C03625=1096.715,71.531,441.280,176.195,16.215,152.221
C03626=1096.709,71.282,441.296,176.193,16.214,152.222
C03627=1096.703,71.032,441.313,176.190,16.213,152.222
C03628=1096.698,70.783,441.330,176.188,16.213,152.222
C03629=1096.692,70.534,441.346,176.185,16.211,152.223
C03630=1096.687,70.284,441.363,176.183,16.211,152.223
C03631=1096.681,70.035,441.380,176.180,16.210,152.223
C03632=1096.675,69.785,441.398,176.179,16.209,152.224
C03633=1096.669,69.536,441.414,176.176,16.209,152.224
C03634=1096.663,69.286,441.431,176.174,16.208,152.224
C03635=1096.657,69.037,441.448,176.172,16.207,152.225
C03636=1096.652,68.787,441.464,176.169,16.206,152.225
C03637=1096.646,68.538,441.481,176.167,16.205,152.225
C03638=1096.641,68.288,441.498,176.164,16.205,152.226
C03639=1096.635,68.039,441.514,176.162,16.204,152.226
C03640=1096.629,67.790,441.531,176.159,16.203,152.226
C03641=1096.623,67.541,441.548,176.157,16.202,152.227
C03642=1096.618,67.291,441.564,176.155,16.201,152.227
C03643=1096.612,67.042,441.581,176.152,16.201,152.227
C03644=1096.606,66.793,441.598,176.150,16.200,152.228
C03645=1096.601,66.543,441.615,176.148,16.199,152.228
C03646=1096.595,66.294,441.631,176.146,16.199,152.228
C03647=1096.590,66.044,441.648,176.143,16.197,152.228
C03648=1096.584,65.795,441.664,176.141,16.197,152.229
C03649=1096.578,65.546,441.680,176.138,16.196,152.229
C03650=1096.572,65.296,441.697,176.136,16.195,152.229
C03651=1096.566,65.047,441.714,176.133,16.194,152.230
C03652=1096.561,64.798,441.731,176.131,16.194,152.230
C03653=1096.555,64.548,441.747,176.129,16.192,152.230
C03654=1096.549,64.299,441.763,176.127,16.192,152.231
C03655=1096.543,64.024,441.782,176.124,16.191,152.231
C03656=1096.537,63.749,441.800,176.122,16.190,152.231
C03657=1096.531,63.475,441.818,176.119,16.189,152.232
C03658=1096.524,63.201,441.836,176.116,16.188,152.232
C03659=1096.519,62.952,441.853,176.114,16.187,152.232
C03660=1096.513,62.702,441.869,176.111,16.186,152.233
C03661=1096.507,62.453,441.885,176.109,16.186,152.233
C03662=1096.501,62.204,441.902,176.107,16.185,152.233
C03663=1096.495,61.954,441.918,176.105,16.184,152.234
C03664=1096.490,61.705,441.935,176.103,16.184,152.234
C03665=1096.484,61.455,441.951,176.100,16.182,152.234
C03666=1096.478,61.206,441.967,176.098,16.182,152.235
C03667=1096.472,60.957,441.983,176.095,16.181,152.235
C03668=1096.466,60.707,442.000,176.093,16.180,152.235
C03669=1096.461,60.458,442.017,176.091,16.179,152.235
C03670=1096.455,60.208,442.033,176.088,16.179,152.236
C03671=1096.449,59.959,442.049,176.086,16.178,152.236
C03672=1096.443,59.709,442.065,176.084,16.177,152.236
C03673=1096.437,59.460,442.082,176.082,16.176,152.237
C03674=1096.432,59.210,442.098,176.079,16.175,152.237
C03675=1096.426,58.961,442.115,176.077,16.174,152.237
C03676=1096.420,58.711,442.130,176.075,16.174,152.238
C03677=1096.414,58.462,442.146,176.072,16.172,152.238
C03678=1096.408,58.212,442.163,176.070,16.172,152.238
C03679=1096.403,57.964,442.179,176.068,16.171,152.239
C03680=1096.397,57.714,442.195,176.066,16.170,152.239
C03681=1096.391,57.465,442.212,176.063,16.169,152.239
C03682=1096.386,57.215,442.228,176.061,16.168,152.239
C03683=1096.380,56.966,442.244,176.059,16.168,152.240
C03684=1096.374,56.716,442.260,176.056,16.167,152.240
C03685=1096.368,56.467,442.276,176.054,16.166,152.240
C03686=1096.362,56.217,442.292,176.052,16.165,152.240
C03687=1096.356,55.968,442.309,176.050,16.164,152.241
C03688=1096.351,55.719,442.325,176.048,16.163,152.241
C03689=1096.346,55.469,442.341,176.045,16.162,152.241
C03690=1096.340,55.220,442.357,176.043,16.161,152.242
C03691=1096.334,54.970,442.373,176.040,16.161,152.242
C03692=1096.328,54.721,442.389,176.038,16.160,152.242
C03693=1096.322,54.472,442.406,176.036,16.159,152.242
C03694=1096.317,54.223,442.421,176.034,16.158,152.243
C03695=1096.311,53.973,442.437,176.032,16.157,152.243
C03696=1096.305,53.724,442.453,176.029,16.156,152.243
C03697=1096.299,53.474,442.469,176.027,16.155,152.244
C03698=1096.294,53.224,442.486,176.025,16.154,152.244
C03699=1096.288,52.975,442.502,176.023,16.153,152.244
C03700=1096.283,52.726,442.518,176.021,16.153,152.244
C03701=1096.277,52.476,442.533,176.018,16.151,152.245
C03702=1096.271,52.227,442.550,176.016,16.151,152.245
C03703=1096.265,51.978,442.566,176.014,16.149,152.245
C03704=1096.260,51.728,442.581,176.011,16.149,152.246
C03705=1096.254,51.479,442.597,176.010,16.148,152.246
C03706=1096.248,51.230,442.614,176.007,16.147,152.246
C03707=1096.243,50.980,442.629,176.005,16.146,152.246
C03708=1096.237,50.730,442.645,176.002,16.145,152.247
C03709=1096.232,50.481,442.661,176.000,16.144,152.247
C03710=1096.226,50.232,442.677,175.999,16.144,152.247
C03711=1096.220,49.982,442.693,175.996,16.142,152.247
C03712=1096.214,49.732,442.709,175.994,16.142,152.248
C03713=1096.209,49.484,442.724,175.991,16.140,152.248
C03714=1096.203,49.234,442.740,175.989,16.140,152.248
C03715=1096.197,48.984,442.756,175.988,16.139,152.248
C03716=1096.191,48.735,442.773,175.985,16.137,152.249
C03717=1096.186,48.486,442.788,175.983,16.137,152.249
C03718=1096.180,48.236,442.804,175.981,16.135,152.249
C03719=1096.174,47.961,442.822,175.979,16.135,152.249
C03720=1096.168,47.687,442.839,175.976,16.133,152.250
C03721=1096.162,47.412,442.857,175.973,16.132,152.250
C03722=1096.156,47.138,442.873,175.971,16.131,152.250
C03723=1096.150,46.888,442.889,175.969,16.130,152.250
C03724=1096.144,46.639,442.905,175.967,16.129,152.251
C03725=1096.139,46.389,442.921,175.965,16.129,152.251
C03726=1096.134,46.139,442.936,175.962,16.127,152.251
C03727=1096.128,45.890,442.952,175.960,16.127,152.251
C03728=1096.122,45.640,442.968,175.958,16.125,152.252
C03729=1096.117,45.391,442.984,175.956,16.125,152.252
C03730=1096.111,45.141,442.999,175.954,16.124,152.252
C03731=1096.105,44.892,443.015,175.951,16.122,152.252
C03732=1096.100,44.643,443.031,175.950,16.122,152.253
C03733=1096.094,44.393,443.047,175.948,16.121,152.253
C03734=1096.089,44.144,443.062,175.945,16.120,152.253
C03735=1096.083,43.894,443.078,175.943,16.119,152.253
C03736=1096.077,43.645,443.094,175.940,16.118,152.254
C03737=1096.072,43.396,443.109,175.939,16.117,152.254
C03738=1096.066,43.146,443.124,175.937,16.116,152.254
C03739=1096.060,42.897,443.140,175.934,16.115,152.254
C03740=1096.055,42.647,443.155,175.932,16.114,152.255
C03741=1096.049,42.398,443.172,175.930,16.112,152.255
C03742=1096.043,42.148,443.187,175.928,16.112,152.255
C03743=1096.038,41.899,443.202,175.926,16.111,152.255
C03744=1096.032,41.650,443.218,175.923,16.110,152.256
C03745=1096.026,41.400,443.234,175.921,16.109,152.256
C03746=1096.021,41.151,443.249,175.919,16.108,152.256
C03747=1096.015,40.901,443.264,175.917,16.107,152.256
C03748=1096.009,40.651,443.280,175.915,16.106,152.256
C03749=1096.004,40.402,443.295,175.913,16.105,152.257
C03750=1095.998,40.152,443.311,175.911,16.104,152.257
C03751=1095.991,39.903,443.326,175.909,16.103,152.257
C03752=1095.986,39.654,443.342,175.906,16.102,152.258
C03753=1095.981,39.404,443.357,175.904,16.101,152.258
C03754=1095.975,39.155,443.372,175.903,16.100,152.258
C03755=1095.969,38.906,443.388,175.900,16.099,152.258
C03756=1095.963,38.656,443.403,175.898,16.098,152.258
C03757=1095.958,38.406,443.419,175.896,16.098,152.259
C03758=1095.952,38.157,443.434,175.893,16.096,152.259
C03759=1095.947,37.908,443.449,175.892,16.095,152.259
C03760=1095.941,37.658,443.465,175.890,16.094,152.259
C03761=1095.934,37.409,443.480,175.887,16.093,152.260
C03762=1095.929,37.159,443.495,175.885,16.092,152.260
C03763=1095.924,36.909,443.511,175.883,16.091,152.260
C03764=1095.918,36.660,443.525,175.881,16.090,152.260
C03765=1095.912,36.411,443.541,175.879,16.089,152.260
C03766=1095.906,36.161,443.556,175.876,16.088,152.261
C03767=1095.900,35.912,443.572,175.875,16.087,152.261
C03768=1095.894,35.662,443.587,175.873,16.087,152.261
C03769=1095.889,35.413,443.602,175.870,16.085,152.262
C03770=1095.883,35.163,443.617,175.868,16.084,152.262
C03771=1095.877,34.914,443.632,175.866,16.083,152.262
C03772=1095.872,34.664,443.647,175.864,16.082,152.262
C03773=1095.866,34.415,443.662,175.862,16.081,152.262
C03774=1095.860,34.166,443.678,175.860,16.081,152.263
C03775=1095.854,33.916,443.693,175.858,16.079,152.263
C03776=1095.849,33.667,443.708,175.856,16.078,152.263
C03777=1095.842,33.417,443.723,175.854,16.078,152.263
C03778=1095.837,33.167,443.739,175.851,16.076,152.264
C03779=1095.831,32.918,443.753,175.850,16.075,152.264
C03780=1095.825,32.668,443.769,175.848,16.074,152.264
C03781=1095.820,32.419,443.784,175.845,16.073,152.264
C03782=1095.814,32.170,443.799,175.843,16.073,152.265
C03783=1095.808,31.895,443.815,175.841,16.071,152.265
C03784=1095.802,31.621,443.832,175.839,16.070,152.265
C03785=1095.795,31.345,443.849,175.836,16.069,152.265
C03786=1095.789,31.071,443.866,175.834,16.068,152.265
C03787=1095.783,30.822,443.880,175.832,16.066,152.266
C03788=1095.778,30.572,443.896,175.830,16.066,152.266
C03789=1095.771,30.323,443.911,175.828,16.065,152.266
C03790=1095.766,30.073,443.926,175.825,16.064,152.266
C03791=1095.760,29.824,443.941,175.824,16.063,152.266
C03792=1095.755,29.574,443.955,175.822,16.062,152.267
C03793=1095.749,29.324,443.970,175.819,16.061,152.267
C03794=1095.744,29.075,443.985,175.818,16.059,152.267
C03795=1095.738,28.826,444.000,175.816,16.059,152.267
C03796=1095.732,28.576,444.015,175.813,16.057,152.268
C03797=1095.727,28.327,444.030,175.811,16.056,152.268
C03798=1095.720,28.077,444.045,175.810,16.056,152.268
C03799=1095.715,27.828,444.060,175.807,16.054,152.268
C03800=1095.709,27.578,444.075,175.805,16.053,152.268
C03801=1095.703,27.329,444.089,175.803,16.052,152.269
C03802=1095.698,27.079,444.104,175.801,16.051,152.269
C03803=1095.692,26.830,444.119,175.799,16.050,152.269
C03804=1095.686,26.580,444.135,175.797,16.049,152.269
C03805=1095.680,26.331,444.149,175.795,16.048,152.270
C03806=1095.674,26.081,444.164,175.793,16.047,152.270
C03807=1095.668,25.832,444.179,175.791,16.046,152.270
C03808=1095.663,25.582,444.194,175.789,16.045,152.270
C03809=1095.657,25.333,444.208,175.787,16.044,152.270
C03810=1095.651,25.083,444.223,175.785,16.043,152.270
C03811=1095.646,24.834,444.238,175.783,16.042,152.271
C03812=1095.640,24.584,444.252,175.781,16.041,152.271
C03813=1095.634,24.335,444.267,175.779,16.040,152.271
C03814=1095.629,24.085,444.282,175.777,16.039,152.271
C03815=1095.622,23.836,444.297,175.774,16.037,152.272
C03816=1095.617,23.586,444.311,175.773,16.037,152.272
C03817=1095.611,23.337,444.326,175.771,16.036,152.272
C03818=1095.605,23.087,444.341,175.768,16.034,152.272
C03819=1095.599,22.838,444.356,175.766,16.034,152.272
C03820=1095.594,22.588,444.370,175.765,16.032,152.272
C03821=1095.589,22.339,444.385,175.763,16.032,152.273
C03822=1095.582,22.089,444.400,175.760,16.030,152.273
C03823=1095.577,21.840,444.414,175.759,16.029,152.273
C03824=1095.570,21.590,444.429,175.757,16.029,152.273
C03825=1095.565,21.341,444.444,175.754,16.027,152.274
C03826=1095.560,21.091,444.458,175.752,16.026,152.274
C03827=1095.553,20.841,444.473,175.751,16.025,152.274
C03828=1095.548,20.592,444.487,175.748,16.024,152.274
C03829=1095.543,20.343,444.502,175.746,16.023,152.274
C03830=1095.537,20.093,444.517,175.745,16.022,152.275
C03831=1095.531,19.844,444.531,175.743,16.021,152.275
C03832=1095.525,19.594,444.546,175.740,16.020,152.275
C03833=1095.519,19.345,444.560,175.738,16.019,152.275
C03834=1095.513,19.095,444.574,175.737,16.018,152.275
C03835=1095.507,18.845,444.589,175.734,16.016,152.276
C03836=1095.502,18.596,444.604,175.732,16.016,152.276
C03837=1095.497,18.347,444.618,175.731,16.014,152.276
C03838=1095.490,18.097,444.633,175.729,16.014,152.276
C03839=1095.485,17.847,444.647,175.726,16.012,152.276
C03840=1095.479,17.598,444.661,175.725,16.011,152.277
C03841=1095.473,17.348,444.676,175.723,16.011,152.277
C03842=1095.467,17.099,444.690,175.720,16.009,152.277
C03843=1095.462,16.850,444.705,175.718,16.008,152.277
C03844=1095.456,16.600,444.720,175.717,16.007,152.277
C03845=1095.450,16.351,444.734,175.715,16.006,152.277
C03846=1095.445,16.101,444.748,175.712,16.004,152.278
C03847=1095.438,15.827,444.764,175.711,16.004,152.278
C03848=1095.431,15.554,444.780,175.708,16.003,152.278
C03849=1095.425,15.281,444.796,175.706,16.001,152.278
C03850=1095.419,15.008,444.812,175.704,16.000,152.279
C03851=1095.413,14.758,444.825,175.702,15.999,152.279
C03852=1095.408,14.509,444.840,175.700,15.998,152.279
C03853=1095.402,14.259,444.854,175.699,15.997,152.279
C03854=1095.396,14.010,444.869,175.696,15.996,152.279
C03855=1095.390,13.760,444.883,175.694,15.995,152.279
C03856=1095.384,13.511,444.898,175.692,15.994,152.280
C03857=1095.378,13.261,444.911,175.690,15.993,152.280
C03858=1095.373,13.012,444.926,175.688,15.991,152.280
C03859=1095.367,12.762,444.940,175.686,15.991,152.280
C03860=1095.361,12.512,444.954,175.685,15.990,152.280
C03861=1095.355,12.263,444.969,175.683,15.989,152.281
C03862=1095.349,12.013,444.982,175.680,15.987,152.281
C03863=1095.343,11.764,444.996,175.678,15.986,152.281
C03864=1095.337,11.515,445.011,175.677,15.986,152.281
C03865=1095.332,11.265,445.025,175.674,15.984,152.281
C03866=1095.325,11.015,445.040,175.672,15.983,152.282
C03867=1095.320,10.766,445.053,175.671,15.982,152.282
C03868=1095.314,10.516,445.067,175.669,15.981,152.282
C03869=1095.308,10.267,445.082,175.666,15.980,152.282
C03870=1095.303,10.017,445.096,175.664,15.979,152.282
C03871=1095.297,9.767,445.110,175.663,15.978,152.282
C03872=1095.291,9.519,445.124,175.661,15.977,152.283
C03873=1095.285,9.269,445.138,175.659,15.975,152.283
C03874=1095.279,9.019,445.152,175.657,15.975,152.283
C03875=1095.274,8.769,445.166,175.655,15.974,152.283
C03876=1095.268,8.520,445.181,175.653,15.973,152.283
C03877=1095.262,8.270,445.195,175.651,15.971,152.284
C03878=1095.256,8.021,445.209,175.649,15.970,152.284
C03879=1095.250,7.771,445.222,175.647,15.969,152.284
C03880=1095.244,7.522,445.236,175.645,15.969,152.284
C03881=1095.238,7.272,445.251,175.644,15.967,152.284
C03882=1095.233,7.023,445.265,175.641,15.966,152.285
C03883=1095.227,6.773,445.278,175.640,15.965,152.285
C03884=1095.221,6.524,445.293,175.638,15.964,152.285
C03885=1095.216,6.274,445.307,175.636,15.963,152.285
C03886=1095.209,6.024,445.320,175.634,15.961,152.285
C03887=1095.204,5.775,445.334,175.632,15.961,152.285
C03888=1095.198,5.525,445.348,175.630,15.959,152.286
C03889=1095.192,5.276,445.363,175.628,15.959,152.286
C03890=1095.187,5.027,445.377,175.626,15.957,152.286
C03891=1095.180,4.777,445.390,175.624,15.956,152.286
C03892=1095.175,4.527,445.404,175.622,15.955,152.286
C03893=1095.169,4.278,445.418,175.621,15.954,152.287
C03894=1095.164,4.028,445.432,175.618,15.953,152.287
C03895=1095.158,3.779,445.446,175.617,15.952,152.287
C03896=1095.152,3.529,445.459,175.615,15.951,152.287
C03897=1095.146,3.280,445.474,175.613,15.950,152.287
C03898=1095.140,3.030,445.488,175.610,15.948,152.287
C03899=1095.135,2.780,445.502,175.609,15.947,152.288
C03900=1095.129,2.531,445.516,175.607,15.946,152.288
C03901=1095.123,2.282,445.529,175.605,15.945,152.288
C03902=1095.118,2.032,445.543,175.604,15.944,152.288
C03903=1095.112,1.782,445.557,175.601,15.943,152.288
C03904=1095.106,1.532,445.571,175.599,15.942,152.288
C03905=1095.100,1.283,445.585,175.598,15.941,152.288
C03906=1095.094,1.033,445.598,175.596,15.940,152.289
C03907=1095.089,0.784,445.612,175.594,15.938,152.289
C03908=1095.083,0.534,445.626,175.592,15.937,152.289
C03909=1095.078,0.285,445.640,175.590,15.936,152.289
C03910=1095.072,0.035,445.653,175.589,15.935,152.289
C03911=1095.065,-0.236,445.668,175.586,15.934,152.290
C03912=1095.059,-0.507,445.683,175.584,15.933,152.290
C03913=1095.053,-0.779,445.698,175.582,15.932,152.290
C03914=1095.047,-1.049,445.713,175.580,15.930,152.290
C03915=1095.041,-1.299,445.727,175.578,15.929,152.290
C03916=1095.035,-1.548,445.740,175.576,15.928,152.290
C03917=1095.029,-1.799,445.754,175.575,15.927,152.291
C03918=1095.024,-2.048,445.768,175.572,15.925,152.291
C03919=1095.018,-2.298,445.781,175.571,15.925,152.291
C03920=1095.012,-2.548,445.795,175.569,15.924,152.291
C03921=1095.007,-2.797,445.808,175.567,15.922,152.291
C03922=1095.001,-3.047,445.822,175.565,15.921,152.291
C03923=1094.995,-3.296,445.836,175.563,15.920,152.292
C03924=1094.990,-3.546,445.849,175.562,15.919,152.292
C03925=1094.984,-3.795,445.863,175.560,15.918,152.292
C03926=1094.978,-4.044,445.877,175.558,15.917,152.292
C03927=1094.972,-4.294,445.890,175.555,15.916,152.292
C03928=1094.966,-4.543,445.904,175.554,15.915,152.292
C03929=1094.961,-4.793,445.917,175.552,15.914,152.293
C03930=1094.954,-5.043,445.931,175.550,15.913,152.293
C03931=1094.949,-5.293,445.944,175.549,15.912,152.293
C03932=1094.943,-5.542,445.958,175.546,15.910,152.293
C03933=1094.937,-5.792,445.972,175.544,15.909,152.293
C03934=1094.931,-6.041,445.985,175.543,15.908,152.293
C03935=1094.925,-6.291,445.999,175.541,15.907,152.294
C03936=1094.919,-6.541,446.011,175.539,15.906,152.294
C03937=1094.914,-6.790,446.025,175.537,15.905,152.294
C03938=1094.908,-7.039,446.038,175.535,15.904,152.294
C03939=1094.902,-7.289,446.052,175.533,15.903,152.294
C03940=1094.896,-7.538,446.065,175.532,15.902,152.294
C03941=1094.890,-7.788,446.078,175.530,15.901,152.294
C03942=1094.885,-8.038,446.092,175.528,15.900,152.295
C03943=1094.878,-8.287,446.105,175.526,15.898,152.295
C03944=1094.873,-8.536,446.119,175.524,15.897,152.295
C03945=1094.867,-8.786,446.132,175.522,15.896,152.295
C03946=1094.862,-9.036,446.145,175.521,15.895,152.295
C03947=1094.855,-9.285,446.159,175.519,15.894,152.296
C03948=1094.850,-9.535,446.173,175.517,15.893,152.296
C03949=1094.844,-9.785,446.185,175.515,15.892,152.296
C03950=1094.838,-10.034,446.198,175.513,15.891,152.296
C03951=1094.832,-10.284,446.212,175.511,15.890,152.296
C03952=1094.826,-10.533,446.225,175.510,15.888,152.296
C03953=1094.821,-10.783,446.239,175.508,15.888,152.297
C03954=1094.815,-11.032,446.252,175.505,15.886,152.297
C03955=1094.810,-11.282,446.265,175.504,15.885,152.297
C03956=1094.803,-11.532,446.278,175.502,15.884,152.297
C03957=1094.797,-11.781,446.292,175.500,15.883,152.297
C03958=1094.792,-12.031,446.305,175.499,15.882,152.297
C03959=1094.786,-12.280,446.318,175.497,15.881,152.297
C03960=1094.780,-12.530,446.332,175.494,15.879,152.298
C03961=1094.774,-12.780,446.344,175.493,15.878,152.298
C03962=1094.768,-13.029,446.358,175.491,15.878,152.298
C03963=1094.763,-13.279,446.372,175.489,15.876,152.298
C03964=1094.757,-13.529,446.384,175.488,15.875,152.298
C03965=1094.751,-13.778,446.398,175.486,15.875,152.298
C03966=1094.745,-14.028,446.411,175.483,15.873,152.299
C03967=1094.739,-14.277,446.424,175.482,15.872,152.299
C03968=1094.734,-14.527,446.438,175.480,15.871,152.299
C03969=1094.728,-14.777,446.450,175.478,15.870,152.299
C03970=1094.722,-15.026,446.464,175.477,15.869,152.299
C03971=1094.716,-15.276,446.477,175.475,15.868,152.299
C03972=1094.710,-15.526,446.490,175.473,15.867,152.299
C03973=1094.704,-15.775,446.503,175.471,15.865,152.300
C03974=1094.698,-16.025,446.516,175.469,15.864,152.300
C03975=1094.692,-16.294,446.530,175.467,15.863,152.300
C03976=1094.686,-16.563,446.544,175.466,15.862,152.300
C03977=1094.680,-16.834,446.558,175.463,15.861,152.300
C03978=1094.674,-17.103,446.572,175.462,15.860,152.300
C03979=1094.667,-17.353,446.585,175.460,15.859,152.301
C03980=1094.662,-17.602,446.598,175.458,15.858,152.301
C03981=1094.655,-17.852,446.611,175.456,15.856,152.301
C03982=1094.650,-18.102,446.624,175.454,15.855,152.301
C03983=1094.644,-18.351,446.638,175.452,15.854,152.301
C03984=1094.638,-18.601,446.650,175.451,15.853,152.301
C03985=1094.632,-18.850,446.663,175.449,15.852,152.302
C03986=1094.626,-19.099,446.676,175.447,15.851,152.302
C03987=1094.620,-19.349,446.689,175.445,15.850,152.302
C03988=1094.615,-19.599,446.702,175.444,15.849,152.302
C03989=1094.609,-19.849,446.715,175.441,15.847,152.302
C03990=1094.603,-20.098,446.728,175.439,15.847,152.303
C03991=1094.597,-20.348,446.740,175.438,15.846,152.303
C03992=1094.591,-20.597,446.754,175.436,15.844,152.303
C03993=1094.585,-20.847,446.766,175.434,15.844,152.303
C03994=1094.580,-21.097,446.779,175.433,15.843,152.303
C03995=1094.574,-21.346,446.792,175.431,15.841,152.303
C03996=1094.568,-21.596,446.805,175.429,15.841,152.303
C03997=1094.562,-21.845,446.818,175.427,15.839,152.304
C03998=1094.556,-22.095,446.831,175.425,15.838,152.304
C03999=1094.550,-22.345,446.843,175.424,15.837,152.304
C04000=1094.545,-22.594,446.857,175.422,15.836,152.304
C04001=1094.539,-22.844,446.870,175.420,15.835,152.304
C04002=1094.534,-23.093,446.882,175.419,15.834,152.304
C04003=1094.527,-23.343,446.895,175.417,15.833,152.304
C04004=1094.521,-23.593,446.908,175.415,15.832,152.305
C04005=1094.516,-23.842,446.920,175.413,15.830,152.305
C04006=1094.509,-24.092,446.933,175.411,15.829,152.305
C04007=1094.503,-24.342,446.946,175.409,15.828,152.305
C04008=1094.498,-24.591,446.958,175.408,15.827,152.305
C04009=1094.493,-24.841,446.971,175.406,15.826,152.305
C04010=1094.487,-25.090,446.985,175.404,15.825,152.306
C04011=1094.481,-25.340,446.997,175.403,15.824,152.306
C04012=1094.475,-25.590,447.010,175.401,15.823,152.306
C04013=1094.470,-25.839,447.022,175.398,15.821,152.306
C04014=1094.463,-26.088,447.035,175.397,15.820,152.306
C04015=1094.457,-26.338,447.048,175.395,15.819,152.306
C04016=1094.452,-26.588,447.060,175.393,15.818,152.306
C04017=1094.446,-26.838,447.073,175.392,15.817,152.307
C04018=1094.440,-27.087,447.086,175.390,15.816,152.307
C04019=1094.434,-27.337,447.098,175.388,15.815,152.307
C04020=1094.428,-27.586,447.111,175.386,15.814,152.307
C04021=1094.422,-27.836,447.123,175.385,15.813,152.307
C04022=1094.416,-28.086,447.136,175.383,15.812,152.307
C04023=1094.411,-28.335,447.149,175.381,15.811,152.308
C04024=1094.405,-28.585,447.161,175.379,15.809,152.308
C04025=1094.399,-28.835,447.174,175.377,15.809,152.308
C04026=1094.393,-29.084,447.187,175.376,15.808,152.308
C04027=1094.387,-29.334,447.199,175.374,15.806,152.308
C04028=1094.382,-29.583,447.211,175.372,15.806,152.308
C04029=1094.375,-29.832,447.224,175.370,15.805,152.308
C04030=1094.369,-30.082,447.237,175.369,15.804,152.309
C04031=1094.363,-30.332,447.249,175.367,15.803,152.309
C04032=1094.357,-30.582,447.262,175.365,15.802,152.309
C04033=1094.352,-30.831,447.274,175.363,15.801,152.309
C04034=1094.346,-31.081,447.286,175.361,15.799,152.309
C04035=1094.340,-31.331,447.299,175.360,15.798,152.309
C04036=1094.334,-31.581,447.311,175.358,15.797,152.310
C04037=1094.329,-31.829,447.324,175.356,15.796,152.310
C04038=1094.323,-32.079,447.337,175.354,15.795,152.310
C04039=1094.316,-32.349,447.350,175.353,15.794,152.310
C04040=1094.310,-32.617,447.363,175.351,15.793,152.310
C04041=1094.303,-32.886,447.376,175.349,15.791,152.310
C04042=1094.297,-33.155,447.390,175.347,15.791,152.311
C04043=1094.291,-33.404,447.402,175.345,15.790,152.311
C04044=1094.285,-33.654,447.415,175.343,15.788,152.311
C04045=1094.279,-33.904,447.427,175.342,15.788,152.311
C04046=1094.274,-34.153,447.440,175.340,15.787,152.311
C04047=1094.267,-34.403,447.452,175.338,15.785,152.311
C04048=1094.261,-34.653,447.464,175.336,15.785,152.312
C04049=1094.256,-34.902,447.476,175.335,15.783,152.312
C04050=1094.250,-35.152,447.489,175.333,15.782,152.312
C04051=1094.244,-35.402,447.501,175.331,15.782,152.312
C04052=1094.239,-35.651,447.514,175.330,15.780,152.312
C04053=1094.232,-35.901,447.526,175.327,15.779,152.312
C04054=1094.226,-36.150,447.538,175.326,15.778,152.313
C04055=1094.221,-36.400,447.551,175.324,15.777,152.313
C04056=1094.215,-36.650,447.563,175.322,15.776,152.313
C04057=1094.209,-36.899,447.575,175.321,15.775,152.313
C04058=1094.203,-37.149,447.588,175.319,15.774,152.313
C04059=1094.197,-37.398,447.600,175.317,15.773,152.313
C04060=1094.191,-37.648,447.612,175.316,15.772,152.313
C04061=1094.186,-37.897,447.624,175.314,15.771,152.314
C04062=1094.180,-38.147,447.637,175.312,15.770,152.314
C04063=1094.175,-38.398,447.649,175.311,15.768,152.314
C04064=1094.169,-38.646,447.660,175.309,15.768,152.314
C04065=1094.163,-38.896,447.673,175.307,15.767,152.314
C04066=1094.157,-39.146,447.685,175.306,15.765,152.314
C04067=1094.150,-39.396,447.697,175.304,15.765,152.314
C04068=1094.145,-39.645,447.710,175.302,15.764,152.315
C04069=1094.139,-39.895,447.722,175.300,15.762,152.315
C04070=1094.132,-40.144,447.734,175.299,15.762,152.315
C04071=1094.127,-40.394,447.746,175.297,15.761,152.315
C04072=1094.121,-40.644,447.758,175.295,15.760,152.315
C04073=1094.115,-40.894,447.770,175.293,15.758,152.315
C04074=1094.109,-41.143,447.782,175.291,15.757,152.316
C04075=1094.103,-41.392,447.794,175.289,15.756,152.316
C04076=1094.097,-41.642,447.807,175.288,15.755,152.316
C04077=1094.092,-41.892,447.818,175.286,15.754,152.316
C04078=1094.085,-42.142,447.830,175.284,15.753,152.316
C04079=1094.079,-42.392,447.843,175.283,15.752,152.316
C04080=1094.074,-42.641,447.855,175.281,15.751,152.317
C04081=1094.067,-42.890,447.867,175.279,15.750,152.317
C04082=1094.062,-43.140,447.878,175.277,15.749,152.317
C04083=1094.056,-43.390,447.890,175.276,15.748,152.317
C04084=1094.050,-43.640,447.903,175.274,15.747,152.317
C04085=1094.044,-43.889,447.915,175.272,15.746,152.317
C04086=1094.038,-44.139,447.926,175.270,15.745,152.318
C04087=1094.032,-44.389,447.939,175.269,15.744,152.318
C04088=1094.026,-44.638,447.950,175.267,15.743,152.318
C04089=1094.020,-44.888,447.963,175.265,15.742,152.318
C04090=1094.015,-45.137,447.974,175.264,15.741,152.318
C04091=1094.009,-45.387,447.986,175.262,15.740,152.318
C04092=1094.003,-45.637,447.999,175.260,15.739,152.318
C04093=1093.997,-45.886,448.010,175.259,15.738,152.319
C04094=1093.991,-46.136,448.022,175.257,15.738,152.319
C04095=1093.985,-46.385,448.034,175.255,15.736,152.319
C04096=1093.979,-46.635,448.047,175.254,15.735,152.319
C04097=1093.973,-46.884,448.057,175.252,15.735,152.319
C04098=1093.967,-47.134,448.070,175.250,15.733,152.319
C04099=1093.962,-47.384,448.083,175.249,15.732,152.320
C04100=1093.956,-47.634,448.093,175.247,15.732,152.320
C04101=1093.950,-47.884,448.106,175.245,15.730,152.320
C04102=1093.944,-48.133,448.117,175.243,15.729,152.320
C04103=1093.938,-48.402,448.130,175.242,15.729,152.320
C04104=1093.932,-48.671,448.143,175.240,15.727,152.320
C04105=1093.925,-48.940,448.156,175.237,15.726,152.321
C04106=1093.919,-49.210,448.168,175.236,15.725,152.321
C04107=1093.913,-49.459,448.180,175.234,15.724,152.321
C04108=1093.908,-49.709,448.192,175.232,15.723,152.321
C04109=1093.901,-49.959,448.204,175.231,15.722,152.321
C04110=1093.895,-50.208,448.216,175.229,15.721,152.321
C04111=1093.889,-50.458,448.227,175.227,15.720,152.322
C04112=1093.883,-50.708,448.240,175.226,15.719,152.322
C04113=1093.878,-50.957,448.251,175.224,15.718,152.322
C04114=1093.871,-51.207,448.262,175.222,15.717,152.322
C04115=1093.866,-51.457,448.274,175.220,15.716,152.322
C04116=1093.859,-51.706,448.286,175.219,15.715,152.322
C04117=1093.853,-51.956,448.298,175.217,15.714,152.323
C04118=1093.848,-52.206,448.309,175.215,15.713,152.323
C04119=1093.841,-52.455,448.321,175.213,15.712,152.323
C04120=1093.835,-52.705,448.332,175.212,15.712,152.323
C04121=1093.829,-52.954,448.344,175.211,15.711,152.323
C04122=1093.824,-53.204,448.356,175.209,15.710,152.323
C04123=1093.817,-53.454,448.368,175.207,15.709,152.324
C04124=1093.811,-53.704,448.379,175.205,15.708,152.324
C04125=1093.805,-53.953,448.390,175.204,15.707,152.324
C04126=1093.799,-54.203,448.402,175.202,15.706,152.324
C04127=1093.793,-54.452,448.414,175.200,15.705,152.324
C04128=1093.787,-54.702,448.425,175.199,15.704,152.324
C04129=1093.781,-54.951,448.437,175.197,15.704,152.325
C04130=1093.775,-55.202,448.449,175.195,15.702,152.325
C04131=1093.769,-55.450,448.460,175.193,15.702,152.325
C04132=1093.763,-55.701,448.471,175.192,15.701,152.325
C04133=1093.758,-55.950,448.483,175.190,15.700,152.325
C04134=1093.751,-56.200,448.495,175.188,15.699,152.325
C04135=1093.745,-56.450,448.506,175.186,15.698,152.326
C04136=1093.739,-56.699,448.518,175.185,15.697,152.326
C04137=1093.732,-56.949,448.529,175.183,15.696,152.326
C04138=1093.727,-57.198,448.541,175.181,15.695,152.326
C04139=1093.721,-57.449,448.552,175.180,15.694,152.326
C04140=1093.715,-57.698,448.563,175.178,15.693,152.327
C04141=1093.708,-57.948,448.575,175.176,15.692,152.327
C04142=1093.703,-58.198,448.587,175.174,15.691,152.327
C04143=1093.697,-58.447,448.597,175.173,15.690,152.327
C04144=1093.691,-58.697,448.609,175.172,15.690,152.327
C04145=1093.685,-58.946,448.620,175.170,15.689,152.327
C04146=1093.678,-59.196,448.632,175.168,15.688,152.328
C04147=1093.673,-59.445,448.644,175.167,15.687,152.328
C04148=1093.667,-59.696,448.655,175.165,15.686,152.328
C04149=1093.661,-59.945,448.667,175.163,15.685,152.328
C04150=1093.655,-60.195,448.678,175.161,15.684,152.328
C04151=1093.649,-60.444,448.689,175.160,15.683,152.328
C04152=1093.643,-60.694,448.701,175.158,15.682,152.329
C04153=1093.637,-60.944,448.712,175.156,15.682,152.329
C04154=1093.631,-61.194,448.723,175.154,15.680,152.329
C04155=1093.625,-61.443,448.734,175.153,15.680,152.329
C04156=1093.619,-61.692,448.746,175.151,15.679,152.329
C04157=1093.613,-61.942,448.757,175.149,15.678,152.330
C04158=1093.608,-62.192,448.769,175.147,15.677,152.330
C04159=1093.601,-62.442,448.780,175.147,15.676,152.330
C04160=1093.595,-62.691,448.791,175.145,15.675,152.330
C04161=1093.589,-62.941,448.803,175.143,15.674,152.330
C04162=1093.583,-63.191,448.814,175.141,15.674,152.330
C04163=1093.578,-63.440,448.824,175.140,15.672,152.330
C04164=1093.572,-63.690,448.837,175.138,15.672,152.331
C04165=1093.566,-63.940,448.848,175.136,15.671,152.331
C04166=1093.560,-64.189,448.859,175.134,15.670,152.331
C04167=1093.554,-64.460,448.871,175.133,15.669,152.331
C04168=1093.547,-64.730,448.883,175.131,15.668,152.331
C04169=1093.541,-65.001,448.896,175.129,15.667,152.332
C04170=1093.534,-65.271,448.907,175.127,15.666,152.332
C04171=1093.529,-65.521,448.919,175.126,15.665,152.332
C04172=1093.522,-65.771,448.930,175.124,15.664,152.332
C04173=1093.516,-66.020,448.942,175.122,15.663,152.332
C04174=1093.511,-66.270,448.953,175.120,15.663,152.333
C04175=1093.504,-66.520,448.964,175.119,15.661,152.333
C04176=1093.498,-66.769,448.975,175.117,15.661,152.333
C04177=1093.493,-67.019,448.986,175.115,15.660,152.333
C04178=1093.486,-67.269,448.997,175.114,15.659,152.333
C04179=1093.481,-67.519,449.008,175.113,15.658,152.333
C04180=1093.475,-67.768,449.020,175.111,15.657,152.333
C04181=1093.469,-68.018,449.031,175.109,15.656,152.334
C04182=1093.463,-68.267,449.042,175.108,15.655,152.334
C04183=1093.457,-68.517,449.053,175.106,15.655,152.334
C04184=1093.451,-68.767,449.064,175.104,15.653,152.334
C04185=1093.445,-69.017,449.075,175.102,15.653,152.334
C04186=1093.440,-69.266,449.086,175.101,15.652,152.335
C04187=1093.433,-69.516,449.097,175.099,15.652,152.335
C04188=1093.428,-69.766,449.108,175.098,15.650,152.335
C04189=1093.422,-70.015,449.119,175.096,15.650,152.335
C04190=1093.416,-70.265,449.130,175.094,15.649,152.335
C04191=1093.410,-70.515,449.141,175.092,15.648,152.336
C04192=1093.404,-70.764,449.152,175.091,15.647,152.336
C04193=1093.399,-71.014,449.164,175.089,15.646,152.336
C04194=1093.392,-71.264,449.175,175.087,15.645,152.336
C04195=1093.387,-71.513,449.186,175.086,15.644,152.336
C04196=1093.381,-71.763,449.197,175.085,15.644,152.336
C04197=1093.375,-72.012,449.208,175.083,15.642,152.336
C04198=1093.369,-72.262,449.219,175.081,15.642,152.337
C04199=1093.363,-72.512,449.230,175.080,15.641,152.337
C04200=1093.357,-72.761,449.241,175.078,15.640,152.337
C04201=1093.352,-73.011,449.252,175.076,15.639,152.337
C04202=1093.345,-73.261,449.263,175.074,15.638,152.337
C04203=1093.340,-73.511,449.273,175.073,15.637,152.338
C04204=1093.334,-73.761,449.284,175.072,15.637,152.338
C04205=1093.328,-74.010,449.295,175.070,15.636,152.338
C04206=1093.322,-74.260,449.306,175.068,15.635,152.338
C04207=1093.316,-74.510,449.317,175.066,15.634,152.338
C04208=1093.311,-74.759,449.328,175.065,15.633,152.338
C04209=1093.305,-75.009,449.339,175.063,15.632,152.339
C04210=1093.298,-75.259,449.350,175.061,15.631,152.339
C04211=1093.292,-75.508,449.360,175.060,15.631,152.339
C04212=1093.286,-75.758,449.371,175.058,15.630,152.339
C04213=1093.280,-76.008,449.383,175.056,15.629,152.339
C04214=1093.274,-76.257,449.393,175.055,15.628,152.340
C04215=1093.268,-76.507,449.404,175.053,15.628,152.340
C04216=1093.263,-76.756,449.415,175.051,15.627,152.340
C04217=1093.256,-77.006,449.426,175.049,15.626,152.340
C04218=1093.250,-77.256,449.436,175.048,15.626,152.340
C04219=1093.244,-77.506,449.447,175.047,15.624,152.341
C04220=1093.239,-77.755,449.458,175.045,15.624,152.341
C04221=1093.232,-78.006,449.469,175.043,15.623,152.341
C04222=1093.226,-78.255,449.479,175.041,15.622,152.341
C04223=1093.220,-78.504,449.490,175.039,15.621,152.341
C04224=1093.214,-78.754,449.501,175.039,15.621,152.341
C04225=1093.208,-79.005,449.512,175.037,15.620,152.342
C04226=1093.203,-79.254,449.522,175.035,15.619,152.342
C04227=1093.197,-79.503,449.533,175.033,15.618,152.342
C04228=1093.190,-79.753,449.544,175.031,15.618,152.342
C04229=1093.184,-80.003,449.555,175.030,15.616,152.342
C04230=1093.178,-80.252,449.566,175.029,15.616,152.343
C04231=1093.172,-80.525,449.577,175.027,15.616,152.343
C04232=1093.165,-80.798,449.588,175.025,15.614,152.343
C04233=1093.158,-81.071,449.600,175.023,15.614,152.343
C04234=1093.152,-81.343,449.612,175.021,15.613,152.344
C04235=1093.146,-81.593,449.622,175.020,15.612,152.344
C04236=1093.139,-81.843,449.633,175.018,15.611,152.344
C04237=1093.133,-82.092,449.644,175.016,15.611,152.344
C04238=1093.128,-82.342,449.654,175.014,15.610,152.345
C04239=1093.121,-82.591,449.665,175.013,15.609,152.345
C04240=1093.115,-82.842,449.675,175.011,15.609,152.345
C04241=1093.109,-83.091,449.686,175.010,15.608,152.345
C04242=1093.103,-83.340,449.696,175.008,15.607,152.345
C04243=1093.097,-83.590,449.707,175.006,15.606,152.345
C04244=1093.090,-83.840,449.717,175.005,15.606,152.346
C04245=1093.085,-84.090,449.728,175.003,15.605,152.346
C04246=1093.079,-84.339,449.739,175.001,15.604,152.346
C04247=1093.073,-84.589,449.748,175.000,15.604,152.346
C04248=1093.067,-84.839,449.759,174.998,15.602,152.346
C04249=1093.061,-85.089,449.771,174.997,15.602,152.347
C04250=1093.054,-85.338,449.781,174.995,15.602,152.347
C04251=1093.049,-85.588,449.791,174.993,15.600,152.347
C04252=1093.042,-85.837,449.801,174.991,15.600,152.347
C04253=1093.037,-86.087,449.812,174.990,15.600,152.347
C04254=1093.031,-86.338,449.823,174.988,15.599,152.348
C04255=1093.024,-86.587,449.833,174.987,15.598,152.348
C04256=1093.018,-86.836,449.844,174.985,15.597,152.348
C04257=1093.012,-87.086,449.853,174.983,15.597,152.348
C04258=1093.006,-87.336,449.864,174.982,15.596,152.348
C04259=1093.000,-87.586,449.874,174.980,15.595,152.349
C04260=1092.994,-87.836,449.885,174.978,15.595,152.349
C04261=1092.988,-88.085,449.896,174.977,15.593,152.349
C04262=1092.982,-88.335,449.906,174.975,15.593,152.349
C04263=1092.976,-88.584,449.916,174.974,15.593,152.350
C04264=1092.970,-88.833,449.927,174.972,15.592,152.350
C04265=1092.964,-89.084,449.937,174.970,15.591,152.350
C04266=1092.957,-89.333,449.948,174.968,15.590,152.350
C04267=1092.952,-89.584,449.958,174.967,15.590,152.350
C04268=1092.946,-89.833,449.969,174.966,15.589,152.351
C04269=1092.940,-90.083,449.978,174.964,15.588,152.351
C04270=1092.934,-90.332,449.989,174.962,15.588,152.351
C04271=1092.928,-90.582,449.999,174.961,15.588,152.351
C04272=1092.922,-90.832,450.010,174.959,15.586,152.351
C04273=1092.915,-91.082,450.020,174.957,15.586,152.352
C04274=1092.910,-91.332,450.030,174.955,15.585,152.352
C04275=1092.903,-91.581,450.041,174.955,15.584,152.352
C04276=1092.898,-91.831,450.051,174.953,15.584,152.352
C04277=1092.891,-92.080,450.061,174.951,15.583,152.353
C04278=1092.886,-92.330,450.071,174.949,15.582,152.353
C04279=1092.879,-92.579,450.081,174.948,15.582,152.353
C04280=1092.874,-92.830,450.092,174.946,15.581,152.353
C04281=1092.868,-93.079,450.102,174.944,15.581,152.353
C04282=1092.862,-93.329,450.112,174.943,15.580,152.354
C04283=1092.855,-93.579,450.123,174.942,15.579,152.354
C04284=1092.850,-93.829,450.133,174.940,15.579,152.354
C04285=1092.843,-94.078,450.143,174.938,15.578,152.354
C04286=1092.838,-94.328,450.153,174.936,15.577,152.355
C04287=1092.831,-94.577,450.164,174.935,15.577,152.355
C04288=1092.826,-94.827,450.174,174.933,15.576,152.355
C04289=1092.819,-95.077,450.184,174.931,15.575,152.355
C04290=1092.814,-95.327,450.194,174.930,15.575,152.355
C04291=1092.808,-95.576,450.204,174.929,15.574,152.355
C04292=1092.802,-95.826,450.215,174.927,15.574,152.356
C04293=1092.796,-96.076,450.224,174.925,15.573,152.356
C04294=1092.790,-96.325,450.235,174.923,15.572,152.356
C04295=1092.783,-96.600,450.246,174.921,15.571,152.356
C04296=1092.776,-96.875,450.258,174.920,15.571,152.357
C04297=1092.771,-97.150,450.268,174.918,15.570,152.357
C04298=1092.763,-97.425,450.280,174.917,15.570,152.357
C04299=1092.758,-97.675,450.290,174.915,15.569,152.357
C04300=1092.751,-97.924,450.300,174.913,15.568,152.358
C04301=1092.745,-98.174,450.310,174.912,15.568,152.358
C04302=1092.740,-98.424,450.320,174.910,15.567,152.358
C04303=1092.733,-98.673,450.330,174.908,15.566,152.358
C04304=1092.727,-98.923,450.340,174.906,15.566,152.359
C04305=1092.721,-99.174,450.350,174.905,15.566,152.359
C04306=1092.715,-99.423,450.360,174.903,15.565,152.359
C04307=1092.709,-99.673,450.370,174.901,15.564,152.359
C04308=1092.702,-99.923,450.380,174.901,15.564,152.359
C04309=1092.697,-100.172,450.390,174.899,15.563,152.360
C04310=1092.690,-100.422,450.400,174.897,15.562,152.360
C04311=1092.684,-100.672,450.410,174.896,15.562,152.360
C04312=1092.679,-100.921,450.420,174.894,15.562,152.360
C04313=1092.672,-101.171,450.430,174.892,15.561,152.361
C04314=1092.666,-101.421,450.440,174.890,15.560,152.361
C04315=1092.660,-101.670,450.450,174.889,15.560,152.361
C04316=1092.654,-101.920,450.460,174.887,15.559,152.361
C04317=1092.648,-102.170,450.470,174.885,15.558,152.361
C04318=1092.642,-102.419,450.480,174.884,15.558,152.362
C04319=1092.636,-102.669,450.490,174.882,15.558,152.362
C04320=1092.630,-102.919,450.500,174.880,15.557,152.362
C04321=1092.624,-103.169,450.509,174.879,15.557,152.362
C04322=1092.617,-103.418,450.519,174.877,15.556,152.363
C04323=1092.612,-103.668,450.530,174.876,15.556,152.363
C04324=1092.606,-103.918,450.539,174.875,15.555,152.363
C04325=1092.600,-104.168,450.549,174.873,15.554,152.363
C04326=1092.593,-104.417,450.559,174.871,15.554,152.364
C04327=1092.588,-104.667,450.569,174.869,15.553,152.364
C04328=1092.581,-104.917,450.579,174.868,15.553,152.364
C04329=1092.575,-105.167,450.588,174.866,15.552,152.364
C04330=1092.569,-105.416,450.598,174.864,15.552,152.365
C04331=1092.563,-105.666,450.608,174.863,15.552,152.365
C04332=1092.557,-105.916,450.618,174.861,15.551,152.365
C04333=1092.551,-106.165,450.628,174.859,15.550,152.365
C04334=1092.545,-106.415,450.638,174.858,15.550,152.366
C04335=1092.539,-106.665,450.647,174.857,15.549,152.366
C04336=1092.532,-106.914,450.657,174.855,15.548,152.366
C04337=1092.527,-107.164,450.668,174.853,15.548,152.366
C04338=1092.521,-107.414,450.677,174.852,15.548,152.366
C04339=1092.514,-107.664,450.687,174.850,15.547,152.367
C04340=1092.508,-107.914,450.696,174.849,15.547,152.367
C04341=1092.502,-108.164,450.706,174.847,15.546,152.367
C04342=1092.496,-108.413,450.716,174.845,15.545,152.367
C04343=1092.489,-108.663,450.726,174.844,15.545,152.368
C04344=1092.484,-108.913,450.736,174.842,15.545,152.368
C04345=1092.478,-109.162,450.745,174.841,15.545,152.368
C04346=1092.472,-109.412,450.755,174.839,15.544,152.368
C04347=1092.466,-109.662,450.765,174.837,15.543,152.369
C04348=1092.459,-109.912,450.774,174.836,15.543,152.369
C04349=1092.453,-110.162,450.784,174.834,15.543,152.369
C04350=1092.447,-110.411,450.793,174.832,15.542,152.369
C04351=1092.441,-110.661,450.803,174.831,15.542,152.370
C04352=1092.434,-110.910,450.813,174.829,15.541,152.370
C04353=1092.428,-111.160,450.823,174.827,15.541,152.370
C04354=1092.422,-111.410,450.832,174.826,15.540,152.370
C04355=1092.416,-111.659,450.841,174.824,15.540,152.371
C04356=1092.410,-111.909,450.851,174.822,15.539,152.371
C04357=1092.405,-112.159,450.861,174.821,15.539,152.371
C04358=1092.399,-112.409,450.871,174.819,15.538,152.371
C04359=1092.391,-112.676,450.881,174.817,15.538,152.372
C04360=1092.385,-112.944,450.891,174.816,15.538,152.372
C04361=1092.379,-113.211,450.902,174.814,15.537,152.372
C04362=1092.372,-113.478,450.912,174.812,15.536,152.373
C04363=1092.366,-113.727,450.921,174.811,15.537,152.373
C04364=1092.359,-113.977,450.931,174.809,15.536,152.373
C04365=1092.354,-114.226,450.940,174.807,15.535,152.373
C04366=1092.348,-114.476,450.950,174.806,15.535,152.374
C04367=1092.341,-114.726,450.959,174.804,15.535,152.374
C04368=1092.335,-114.976,450.969,174.802,15.534,152.374
C04369=1092.329,-115.226,450.978,174.801,15.534,152.374
C04370=1092.323,-115.475,450.988,174.799,15.533,152.375
C04371=1092.317,-115.725,450.998,174.798,15.533,152.375
C04372=1092.311,-115.975,451.007,174.796,15.533,152.375
C04373=1092.304,-116.225,451.017,174.794,15.532,152.375
C04374=1092.298,-116.475,451.026,174.793,15.532,152.376
C04375=1092.292,-116.724,451.036,174.791,15.531,152.376
C04376=1092.286,-116.974,451.045,174.790,15.531,152.376
C04377=1092.280,-117.223,451.055,174.788,15.530,152.376
C04378=1092.274,-117.474,451.063,174.786,15.530,152.377
C04379=1092.268,-117.723,451.073,174.785,15.530,152.377
C04380=1092.262,-117.973,451.083,174.783,15.530,152.377
C04381=1092.256,-118.223,451.092,174.782,15.529,152.378
C04382=1092.250,-118.473,451.102,174.780,15.529,152.378
C04383=1092.243,-118.722,451.111,174.778,15.528,152.378
C04384=1092.237,-118.972,451.120,174.777,15.528,152.378
C04385=1092.231,-119.222,451.130,174.775,15.527,152.379
C04386=1092.225,-119.471,451.139,174.774,15.527,152.379
C04387=1092.219,-119.721,451.149,174.772,15.527,152.379
C04388=1092.213,-119.971,451.158,174.770,15.526,152.380
C04389=1092.207,-120.221,451.167,174.769,15.526,152.380
C04390=1092.201,-120.471,451.177,174.767,15.526,152.380
C04391=1092.194,-120.721,451.186,174.766,15.526,152.380
C04392=1092.188,-120.970,451.195,174.764,15.525,152.381
C04393=1092.182,-121.219,451.204,174.763,15.525,152.381
C04394=1092.176,-121.469,451.214,174.761,15.525,152.381
C04395=1092.170,-121.719,451.223,174.759,15.524,152.381
C04396=1092.164,-121.969,451.232,174.758,15.524,152.382
C04397=1092.158,-122.219,451.242,174.756,15.523,152.382
C04398=1092.151,-122.469,451.251,174.755,15.523,152.382
C04399=1092.144,-122.718,451.260,174.753,15.523,152.382
C04400=1092.139,-122.967,451.270,174.751,15.522,152.383
C04401=1092.133,-123.218,451.278,174.749,15.522,152.383
C04402=1092.127,-123.468,451.288,174.747,15.522,152.383
C04403=1092.121,-123.717,451.298,174.746,15.522,152.384
C04404=1092.115,-123.967,451.307,174.744,15.521,152.384
C04405=1092.108,-124.217,451.316,174.743,15.521,152.384
C04406=1092.102,-124.466,451.325,174.741,15.521,152.384
C04407=1092.096,-124.716,451.334,174.740,15.521,152.385
C04408=1092.090,-124.966,451.344,174.738,15.520,152.385
C04409=1092.084,-125.216,451.353,174.736,15.519,152.385
C04410=1092.077,-125.465,451.362,174.735,15.519,152.385
C04411=1092.071,-125.716,451.371,174.733,15.519,152.386
C04412=1092.065,-125.965,451.380,174.732,15.519,152.386
C04413=1092.059,-126.215,451.390,174.730,15.518,152.386
C04414=1092.052,-126.464,451.399,174.729,15.518,152.387
C04415=1092.047,-126.715,451.408,174.727,15.518,152.387
C04416=1092.040,-126.964,451.417,174.726,15.518,152.387
C04417=1092.034,-127.213,451.426,174.724,15.517,152.388
C04418=1092.028,-127.464,451.435,174.722,15.517,152.388
C04419=1092.022,-127.723,451.444,174.720,15.517,152.388
C04420=1092.016,-127.983,451.454,174.718,15.517,152.388
C04421=1092.010,-128.242,451.464,174.718,15.516,152.389
C04422=1092.015,-128.499,451.476,174.717,15.513,152.388
C04423=1091.609,-128.520,451.359,174.673,15.620,152.418
C04424=1091.604,-128.263,451.347,174.674,15.624,152.418
C04425=1091.608,-128.004,451.337,174.675,15.624,152.418
C04426=1091.615,-127.744,451.327,174.677,15.625,152.418
C04427=1091.620,-127.485,451.318,174.679,15.625,152.418
C04428=1091.627,-127.236,451.308,174.680,15.625,152.417
C04429=1091.634,-126.986,451.299,174.682,15.626,152.417
C04430=1091.639,-126.736,451.290,174.683,15.626,152.417
C04431=1091.646,-126.486,451.281,174.685,15.627,152.417
C04432=1091.652,-126.237,451.272,174.686,15.626,152.416
C04433=1091.658,-125.987,451.263,174.688,15.627,152.416
C04434=1091.664,-125.737,451.254,174.689,15.627,152.416
C04435=1091.670,-125.487,451.244,174.691,15.627,152.415
C04436=1091.677,-125.238,451.235,174.693,15.628,152.415
C04437=1091.683,-124.988,451.226,174.694,15.628,152.415
C04438=1091.689,-124.738,451.216,174.697,15.628,152.414
C04439=1091.695,-124.488,451.208,174.698,15.628,152.414
C04440=1091.701,-124.239,451.198,174.700,15.629,152.414
C04441=1091.708,-123.989,451.189,174.701,15.629,152.414
C04442=1091.714,-123.739,451.180,174.703,15.630,152.413
C04443=1091.720,-123.489,451.171,174.704,15.630,152.413
C04444=1091.725,-123.240,451.161,174.706,15.630,152.413
C04445=1091.732,-122.990,451.152,174.708,15.631,152.413
C04446=1091.738,-122.740,451.142,174.709,15.631,152.412
C04447=1091.745,-122.491,451.133,174.711,15.631,152.412
C04448=1091.750,-122.240,451.125,174.712,15.631,152.412
C04449=1091.757,-121.990,451.115,174.714,15.632,152.412
C04450=1091.763,-121.741,451.105,174.716,15.633,152.411
C04451=1091.768,-121.492,451.096,174.717,15.633,152.411
C04452=1091.775,-121.242,451.087,174.719,15.633,152.411
C04453=1091.781,-120.992,451.078,174.720,15.633,152.410
C04454=1091.788,-120.743,451.068,174.722,15.634,152.410
C04455=1091.793,-120.492,451.059,174.724,15.634,152.410
C04456=1091.800,-120.242,451.050,174.725,15.634,152.410
C04457=1091.806,-119.992,451.040,174.727,15.635,152.409
C04458=1091.811,-119.743,451.031,174.728,15.635,152.409
C04459=1091.818,-119.494,451.021,174.730,15.636,152.409
C04460=1091.824,-119.244,451.012,174.732,15.636,152.409
C04461=1091.830,-118.994,451.002,174.733,15.637,152.408
C04462=1091.837,-118.745,450.993,174.735,15.637,152.408
C04463=1091.843,-118.494,450.984,174.736,15.637,152.408
C04464=1091.849,-118.244,450.975,174.738,15.638,152.408
C04465=1091.855,-117.995,450.965,174.740,15.639,152.407
C04466=1091.861,-117.745,450.956,174.741,15.638,152.407
C04467=1091.867,-117.496,450.946,174.743,15.639,152.407
C04468=1091.873,-117.246,450.937,174.744,15.639,152.407
C04469=1091.879,-116.996,450.927,174.746,15.639,152.406
C04470=1091.885,-116.746,450.918,174.748,15.640,152.406
C04471=1091.891,-116.496,450.908,174.749,15.640,152.406
C04472=1091.898,-116.247,450.899,174.751,15.641,152.406
C04473=1091.904,-115.997,450.889,174.752,15.641,152.405
C04474=1091.910,-115.747,450.879,174.754,15.642,152.405
C04475=1091.916,-115.497,450.870,174.756,15.642,152.405
C04476=1091.922,-115.248,450.861,174.757,15.642,152.405
C04477=1091.928,-114.998,450.851,174.759,15.643,152.404
C04478=1091.934,-114.749,450.842,174.761,15.644,152.404
C04479=1091.940,-114.499,450.832,174.762,15.644,152.404
C04480=1091.946,-114.249,450.822,174.764,15.644,152.403
C04481=1091.953,-113.999,450.813,174.765,15.644,152.403
C04482=1091.959,-113.749,450.803,174.767,15.645,152.403
C04483=1091.965,-113.500,450.794,174.769,15.646,152.403
C04484=1091.972,-113.232,450.784,174.770,15.646,152.403
C04485=1091.978,-112.965,450.774,174.772,15.646,152.402
C04486=1091.984,-112.697,450.764,174.774,15.647,152.402
C04487=1091.991,-112.430,450.753,174.776,15.648,152.402
C04488=1091.997,-112.180,450.743,174.777,15.648,152.401
C04489=1092.003,-111.930,450.734,174.779,15.649,152.401
C04490=1092.009,-111.680,450.724,174.780,15.649,152.401
C04491=1092.016,-111.431,450.715,174.782,15.649,152.401
C04492=1092.022,-111.181,450.705,174.783,15.650,152.400
C04493=1092.028,-110.931,450.695,174.785,15.651,152.400
C04494=1092.034,-110.681,450.686,174.786,15.651,152.400
C04495=1092.040,-110.431,450.676,174.788,15.651,152.400
C04496=1092.046,-110.182,450.667,174.790,15.652,152.399
C04497=1092.053,-109.932,450.657,174.791,15.652,152.399
C04498=1092.058,-109.682,450.646,174.793,15.653,152.399
C04499=1092.064,-109.432,450.637,174.795,15.653,152.399
C04500=1092.071,-109.183,450.627,174.796,15.654,152.399
C04501=1092.077,-108.933,450.618,174.798,15.655,152.398
C04502=1092.083,-108.683,450.608,174.799,15.655,152.398
C04503=1092.089,-108.433,450.598,174.801,15.655,152.398
C04504=1092.095,-108.183,450.589,174.803,15.656,152.398
C04505=1092.102,-107.934,450.579,174.804,15.656,152.397
C04506=1092.108,-107.684,450.569,174.806,15.657,152.397
C04507=1092.113,-107.434,450.559,174.808,15.657,152.397
C04508=1092.120,-107.185,450.549,174.809,15.657,152.397
C04509=1092.126,-106.935,450.540,174.811,15.658,152.396
C04510=1092.132,-106.685,450.530,174.813,15.659,152.396
C04511=1092.138,-106.435,450.521,174.814,15.660,152.396
C04512=1092.145,-106.186,450.510,174.815,15.660,152.396
C04513=1092.150,-105.936,450.500,174.817,15.661,152.395
C04514=1092.156,-105.687,450.491,174.819,15.661,152.395
C04515=1092.162,-105.437,450.481,174.820,15.661,152.395
C04516=1092.168,-105.187,450.472,174.822,15.662,152.395
C04517=1092.174,-104.938,450.461,174.824,15.663,152.394
C04518=1092.180,-104.688,450.451,174.825,15.663,152.394
C04519=1092.186,-104.438,450.442,174.827,15.664,152.394
C04520=1092.192,-104.188,450.432,174.829,15.665,152.394
C04521=1092.199,-103.939,450.422,174.830,15.665,152.394
C04522=1092.204,-103.689,450.412,174.832,15.665,152.393
C04523=1092.210,-103.439,450.402,174.834,15.666,152.393
C04524=1092.216,-103.189,450.393,174.835,15.666,152.393
C04525=1092.223,-102.940,450.382,174.836,15.667,152.393
C04526=1092.228,-102.690,450.372,174.838,15.668,152.393
C04527=1092.235,-102.440,450.362,174.840,15.668,152.392
C04528=1092.241,-102.190,450.353,174.841,15.669,152.392
C04529=1092.247,-101.940,450.342,174.843,15.669,152.392
C04530=1092.253,-101.691,450.332,174.845,15.670,152.391
C04531=1092.259,-101.441,450.323,174.846,15.670,152.391
C04532=1092.266,-101.192,450.312,174.848,15.671,152.391
C04533=1092.271,-100.941,450.302,174.850,15.672,152.391
C04534=1092.277,-100.692,450.293,174.851,15.672,152.391
C04535=1092.284,-100.443,450.282,174.853,15.673,152.390
C04536=1092.290,-100.193,450.273,174.854,15.674,152.390
C04537=1092.296,-99.943,450.263,174.856,15.674,152.390
C04538=1092.302,-99.693,450.252,174.857,15.674,152.390
C04539=1092.308,-99.444,450.243,174.859,15.675,152.390
C04540=1092.314,-99.194,450.233,174.861,15.676,152.389
C04541=1092.320,-98.944,450.222,174.862,15.676,152.389
C04542=1092.326,-98.695,450.213,174.864,15.677,152.389
C04543=1092.332,-98.444,450.203,174.866,15.678,152.389
C04544=1092.338,-98.195,450.192,174.867,15.678,152.388
C04545=1092.344,-97.945,450.183,174.869,15.678,152.388
C04546=1092.350,-97.695,450.172,174.870,15.679,152.388
C04547=1092.357,-97.445,450.162,174.872,15.680,152.388
C04548=1092.363,-97.171,450.151,174.874,15.681,152.388
C04549=1092.370,-96.896,450.140,174.876,15.681,152.387
C04550=1092.376,-96.620,450.129,174.878,15.682,152.387
C04551=1092.382,-96.345,450.118,174.879,15.683,152.387
C04552=1092.389,-96.096,450.107,174.880,15.683,152.387
C04553=1092.394,-95.846,450.097,174.882,15.684,152.386
C04554=1092.401,-95.596,450.087,174.884,15.685,152.386
C04555=1092.406,-95.346,450.077,174.885,15.685,152.386
C04556=1092.413,-95.097,450.066,174.887,15.686,152.386
C04557=1092.419,-94.847,450.057,174.889,15.687,152.386
C04558=1092.424,-94.597,450.047,174.890,15.688,152.385
C04559=1092.431,-94.348,450.036,174.892,15.688,152.385
C04560=1092.436,-94.098,450.026,174.893,15.689,152.385
C04561=1092.443,-93.849,450.016,174.895,15.690,152.385
C04562=1092.449,-93.598,450.005,174.897,15.690,152.385
C04563=1092.455,-93.349,449.995,174.898,15.690,152.384
C04564=1092.461,-93.099,449.985,174.900,15.692,152.384
C04565=1092.466,-92.849,449.974,174.902,15.692,152.384
C04566=1092.473,-92.599,449.965,174.903,15.693,152.384
C04567=1092.478,-92.350,449.954,174.904,15.693,152.384
C04568=1092.485,-92.100,449.944,174.906,15.694,152.383
C04569=1092.490,-91.851,449.933,174.908,15.695,152.383
C04570=1092.496,-91.601,449.924,174.910,15.696,152.383
C04571=1092.502,-91.351,449.913,174.912,15.697,152.383
C04572=1092.508,-91.101,449.903,174.913,15.697,152.383
C04573=1092.515,-90.851,449.892,174.915,15.697,152.382
C04574=1092.521,-90.602,449.882,174.916,15.698,152.382
C04575=1092.527,-90.352,449.872,174.918,15.699,152.382
C04576=1092.533,-90.103,449.861,174.919,15.699,152.382
C04577=1092.539,-89.853,449.851,174.921,15.700,152.382
C04578=1092.545,-89.604,449.841,174.923,15.701,152.381
C04579=1092.550,-89.353,449.831,174.924,15.702,152.381
C04580=1092.557,-89.103,449.819,174.925,15.702,152.381
C04581=1092.563,-88.854,449.809,174.927,15.703,152.381
C04582=1092.569,-88.604,449.799,174.929,15.704,152.381
C04583=1092.575,-88.355,449.789,174.931,15.705,152.380
C04584=1092.581,-88.105,449.778,174.933,15.705,152.380
C04585=1092.587,-87.855,449.768,174.933,15.706,152.380
C04586=1092.593,-87.606,449.757,174.935,15.707,152.380
C04587=1092.599,-87.355,449.747,174.937,15.707,152.379
C04588=1092.605,-87.106,449.737,174.939,15.708,152.379
C04589=1092.611,-86.856,449.726,174.941,15.709,152.379
C04590=1092.617,-86.607,449.716,174.942,15.709,152.379
C04591=1092.623,-86.357,449.705,174.943,15.710,152.379
C04592=1092.630,-86.107,449.695,174.945,15.711,152.379
C04593=1092.635,-85.857,449.684,174.947,15.712,152.378
C04594=1092.641,-85.608,449.674,174.949,15.713,152.378
C04595=1092.648,-85.359,449.663,174.950,15.713,152.378
C04596=1092.653,-85.108,449.653,174.952,15.714,152.378
C04597=1092.660,-84.859,449.642,174.953,15.715,152.378
C04598=1092.666,-84.609,449.632,174.955,15.715,152.377
C04599=1092.671,-84.359,449.621,174.957,15.717,152.377
C04600=1092.678,-84.110,449.611,174.958,15.717,152.377
C04601=1092.684,-83.860,449.600,174.960,15.717,152.377
C04602=1092.690,-83.610,449.589,174.962,15.719,152.377
C04603=1092.696,-83.360,449.579,174.963,15.719,152.376
C04604=1092.702,-83.111,449.569,174.965,15.720,152.376
C04605=1092.708,-82.862,449.558,174.966,15.720,152.376
C04606=1092.715,-82.611,449.547,174.968,15.721,152.376
C04607=1092.720,-82.361,449.537,174.970,15.722,152.376
C04608=1092.727,-82.112,449.527,174.972,15.723,152.375
C04609=1092.732,-81.863,449.516,174.973,15.724,152.375
C04610=1092.739,-81.612,449.504,174.974,15.724,152.375
C04611=1092.745,-81.363,449.495,174.976,15.725,152.375
C04612=1092.752,-81.091,449.483,174.978,15.725,152.375
C04613=1092.758,-80.817,449.471,174.980,15.727,152.374
C04614=1092.764,-80.545,449.459,174.982,15.727,152.374
C04615=1092.771,-80.271,449.448,174.983,15.728,152.374
C04616=1092.778,-80.022,449.437,174.985,15.729,152.374
C04617=1092.784,-79.773,449.427,174.987,15.730,152.374
C04618=1092.789,-79.523,449.416,174.989,15.731,152.373
C04619=1092.795,-79.272,449.405,174.990,15.732,152.373
C04620=1092.801,-79.023,449.394,174.991,15.732,152.373
C04621=1092.808,-78.774,449.384,174.993,15.733,152.373
C04622=1092.813,-78.524,449.373,174.995,15.734,152.373
C04623=1092.820,-78.274,449.362,174.997,15.735,152.372
C04624=1092.825,-78.024,449.351,174.998,15.736,152.372
C04625=1092.831,-77.775,449.340,175.000,15.736,152.372
C04626=1092.837,-77.525,449.330,175.001,15.737,152.372
C04627=1092.844,-77.275,449.319,175.003,15.738,152.372
C04628=1092.849,-77.025,449.308,175.004,15.739,152.372
C04629=1092.855,-76.776,449.298,175.006,15.740,152.371
C04630=1092.861,-76.526,449.287,175.008,15.741,152.371
C04631=1092.867,-76.276,449.275,175.010,15.741,152.371
C04632=1092.873,-76.027,449.265,175.012,15.742,152.371
C04633=1092.879,-75.778,449.254,175.013,15.743,152.371
C04634=1092.885,-75.528,449.243,175.014,15.743,152.370
C04635=1092.892,-75.278,449.232,175.016,15.744,152.370
C04636=1092.897,-75.028,449.221,175.018,15.745,152.370
C04637=1092.903,-74.779,449.210,175.020,15.746,152.370
C04638=1092.909,-74.528,449.200,175.021,15.747,152.370
C04639=1092.915,-74.279,449.189,175.023,15.748,152.370
C04640=1092.920,-74.029,449.178,175.024,15.748,152.369
C04641=1092.926,-73.780,449.167,175.026,15.749,152.369
C04642=1092.933,-73.529,449.156,175.027,15.751,152.369
C04643=1092.938,-73.280,449.145,175.029,15.751,152.369
C04644=1092.944,-73.031,449.134,175.031,15.752,152.369
C04645=1092.950,-72.781,449.123,175.033,15.753,152.369
C04646=1092.956,-72.531,449.112,175.034,15.754,152.368
C04647=1092.962,-72.281,449.101,175.036,15.755,152.368
C04648=1092.968,-72.032,449.090,175.038,15.756,152.368
C04649=1092.973,-71.782,449.080,175.039,15.757,152.368
C04650=1092.980,-71.532,449.068,175.040,15.757,152.368
C04651=1092.985,-71.283,449.057,175.042,15.758,152.368
C04652=1092.991,-71.033,449.047,175.044,15.759,152.367
C04653=1092.998,-70.783,449.035,175.046,15.760,152.367
C04654=1093.003,-70.533,449.024,175.047,15.761,152.367
C04655=1093.009,-70.284,449.014,175.049,15.762,152.367
C04656=1093.015,-70.035,449.003,175.051,15.763,152.367
C04657=1093.021,-69.785,448.991,175.053,15.764,152.367
C04658=1093.027,-69.535,448.980,175.053,15.764,152.366
C04659=1093.033,-69.286,448.969,175.055,15.765,152.366
C04660=1093.038,-69.035,448.957,175.057,15.766,152.366
C04661=1093.044,-68.786,448.946,175.058,15.767,152.366
C04662=1093.050,-68.536,448.935,175.060,15.768,152.366
C04663=1093.056,-68.286,448.924,175.062,15.769,152.366
C04664=1093.062,-68.037,448.913,175.064,15.770,152.365
C04665=1093.068,-67.787,448.902,175.065,15.771,152.365
C04666=1093.074,-67.537,448.891,175.067,15.772,152.365
C04667=1093.080,-67.288,448.880,175.069,15.773,152.365
C04668=1093.086,-67.039,448.869,175.070,15.774,152.365
C04669=1093.092,-66.789,448.857,175.072,15.774,152.365
C04670=1093.097,-66.539,448.846,175.073,15.775,152.364
C04671=1093.103,-66.289,448.835,175.075,15.776,152.364
C04672=1093.109,-66.039,448.824,175.077,15.777,152.364
C04673=1093.115,-65.790,448.813,175.078,15.778,152.364
C04674=1093.121,-65.541,448.801,175.080,15.779,152.364
C04675=1093.127,-65.291,448.790,175.082,15.780,152.364
C04676=1093.134,-65.020,448.778,175.083,15.781,152.364
C04677=1093.140,-64.749,448.766,175.085,15.782,152.363
C04678=1093.146,-64.479,448.754,175.087,15.783,152.363
C04679=1093.152,-64.208,448.742,175.089,15.784,152.363
C04680=1093.159,-63.958,448.731,175.090,15.785,152.363
C04681=1093.165,-63.709,448.719,175.092,15.786,152.363
C04682=1093.171,-63.459,448.708,175.094,15.787,152.362
C04683=1093.177,-63.209,448.697,175.096,15.788,152.362
C04684=1093.182,-62.960,448.685,175.097,15.789,152.362
C04685=1093.188,-62.710,448.673,175.099,15.790,152.362
C04686=1093.194,-62.461,448.663,175.101,15.790,152.362
C04687=1093.201,-62.210,448.651,175.102,15.792,152.362
C04688=1093.206,-61.961,448.640,175.104,15.793,152.361
C04689=1093.212,-61.712,448.629,175.105,15.793,152.361
C04690=1093.218,-61.462,448.617,175.107,15.794,152.361
C04691=1093.224,-61.212,448.606,175.108,15.795,152.361
C04692=1093.230,-60.962,448.594,175.110,15.796,152.361
C04693=1093.236,-60.713,448.583,175.112,15.797,152.361
C04694=1093.242,-60.463,448.572,175.114,15.798,152.360
C04695=1093.248,-60.214,448.560,175.115,15.799,152.360
C04696=1093.254,-59.963,448.549,175.117,15.800,152.360
C04697=1093.260,-59.714,448.538,175.119,15.801,152.360
C04698=1093.266,-59.464,448.526,175.120,15.802,152.360
C04699=1093.272,-59.215,448.515,175.122,15.802,152.360
C04700=1093.277,-58.965,448.503,175.124,15.804,152.359
C04701=1093.284,-58.715,448.492,175.126,15.805,152.359
C04702=1093.290,-58.466,448.481,175.127,15.805,152.359
C04703=1093.296,-58.216,448.469,175.129,15.807,152.359
C04704=1093.302,-57.967,448.458,175.131,15.807,152.359
C04705=1093.308,-57.716,448.446,175.133,15.808,152.359
C04706=1093.313,-57.467,448.435,175.134,15.810,152.359
C04707=1093.320,-57.217,448.423,175.136,15.810,152.358
C04708=1093.326,-56.968,448.412,175.137,15.811,152.358
C04709=1093.332,-56.718,448.400,175.138,15.812,152.358
C04710=1093.337,-56.468,448.389,175.140,15.813,152.358
C04711=1093.344,-56.219,448.377,175.142,15.814,152.358
C04712=1093.350,-55.969,448.366,175.144,15.815,152.357
C04713=1093.356,-55.719,448.355,175.145,15.816,152.357
C04714=1093.361,-55.470,448.343,175.147,15.817,152.357
C04715=1093.368,-55.220,448.331,175.149,15.818,152.357
C04716=1093.374,-54.970,448.319,175.151,15.819,152.357
C04717=1093.380,-54.721,448.308,175.152,15.819,152.357
C04718=1093.386,-54.471,448.296,175.154,15.821,152.357
C04719=1093.392,-54.221,448.285,175.156,15.822,152.356
C04720=1093.398,-53.972,448.273,175.158,15.822,152.356
C04721=1093.403,-53.722,448.262,175.159,15.824,152.356
C04722=1093.410,-53.472,448.250,175.161,15.824,152.356
C04723=1093.416,-53.223,448.239,175.163,15.825,152.356
C04724=1093.422,-52.973,448.227,175.164,15.827,152.356
C04725=1093.428,-52.723,448.215,175.166,15.827,152.355
C04726=1093.434,-52.474,448.203,175.168,15.828,152.355
C04727=1093.440,-52.224,448.192,175.169,15.830,152.355
C04728=1093.446,-51.975,448.180,175.171,15.830,152.355
C04729=1093.452,-51.724,448.169,175.173,15.831,152.355
C04730=1093.458,-51.476,448.157,175.175,15.832,152.355
C04731=1093.465,-51.226,448.145,175.176,15.833,152.354
C04732=1093.470,-50.976,448.133,175.178,15.834,152.354
C04733=1093.476,-50.727,448.122,175.180,15.835,152.354
C04734=1093.483,-50.476,448.110,175.181,15.836,152.354
C04735=1093.488,-50.227,448.098,175.183,15.837,152.354
C04736=1093.494,-49.977,448.087,175.185,15.838,152.354
C04737=1093.500,-49.728,448.075,175.186,15.839,152.353
C04738=1093.506,-49.478,448.063,175.188,15.840,152.353
C04739=1093.511,-49.229,448.051,175.190,15.841,152.353
C04740=1093.518,-48.959,448.038,175.192,15.842,152.353
C04741=1093.524,-48.689,448.026,175.193,15.843,152.353
C04742=1093.530,-48.420,448.013,175.195,15.844,152.353
C04743=1093.537,-48.151,448.000,175.197,15.845,152.353
C04744=1093.543,-47.901,447.988,175.198,15.846,152.352
C04745=1093.549,-47.652,447.976,175.200,15.847,152.352
C04746=1093.555,-47.402,447.964,175.202,15.848,152.352
C04747=1093.560,-47.153,447.953,175.203,15.849,152.352
C04748=1093.566,-46.903,447.940,175.206,15.851,152.352
C04749=1093.572,-46.654,447.929,175.207,15.852,152.352
C04750=1093.578,-46.403,447.917,175.209,15.853,152.351
C04751=1093.584,-46.154,447.905,175.211,15.854,152.351
C04752=1093.590,-45.905,447.893,175.212,15.855,152.351
C04753=1093.596,-45.654,447.881,175.214,15.856,152.351
C04754=1093.601,-45.405,447.869,175.216,15.857,152.351
C04755=1093.608,-45.156,447.857,175.217,15.858,152.351
C04756=1093.614,-44.905,447.845,175.219,15.859,152.351
C04757=1093.619,-44.656,447.833,175.221,15.860,152.350
C04758=1093.626,-44.406,447.821,175.223,15.861,152.350
C04759=1093.631,-44.157,447.809,175.224,15.862,152.350
C04760=1093.637,-43.907,447.798,175.226,15.863,152.350
C04761=1093.643,-43.657,447.785,175.228,15.864,152.350
C04762=1093.648,-43.408,447.773,175.229,15.865,152.350
C04763=1093.655,-43.158,447.761,175.231,15.867,152.350
C04764=1093.661,-42.908,447.749,175.233,15.867,152.349
C04765=1093.667,-42.659,447.738,175.234,15.868,152.349
C04766=1093.673,-42.409,447.725,175.236,15.870,152.349
C04767=1093.678,-42.160,447.713,175.238,15.870,152.349
C04768=1093.685,-41.910,447.701,175.239,15.871,152.349
C04769=1093.690,-41.660,447.689,175.241,15.873,152.349
C04770=1093.695,-41.411,447.677,175.243,15.874,152.349
C04771=1093.702,-41.161,447.665,175.245,15.874,152.348
C04772=1093.708,-40.911,447.652,175.246,15.876,152.348
C04773=1093.714,-40.662,447.641,175.248,15.877,152.348
C04774=1093.720,-40.412,447.628,175.250,15.877,152.348
C04775=1093.726,-40.162,447.617,175.251,15.879,152.348
C04776=1093.732,-39.913,447.605,175.253,15.880,152.348
C04777=1093.738,-39.663,447.592,175.255,15.880,152.347
C04778=1093.743,-39.413,447.580,175.256,15.882,152.347
C04779=1093.750,-39.164,447.568,175.259,15.883,152.347
C04780=1093.755,-38.915,447.556,175.260,15.884,152.347
C04781=1093.761,-38.665,447.543,175.262,15.885,152.347
C04782=1093.768,-38.415,447.531,175.264,15.886,152.347
C04783=1093.773,-38.166,447.519,175.265,15.887,152.347
C04784=1093.779,-37.915,447.507,175.267,15.889,152.347
C04785=1093.785,-37.666,447.495,175.269,15.889,152.346
C04786=1093.790,-37.416,447.482,175.270,15.890,152.346
C04787=1093.797,-37.167,447.470,175.272,15.892,152.346
C04788=1093.803,-36.917,447.458,175.274,15.893,152.346
C04789=1093.808,-36.668,447.446,175.276,15.893,152.346
C04790=1093.814,-36.418,447.433,175.277,15.895,152.346
C04791=1093.820,-36.168,447.421,175.279,15.896,152.346
C04792=1093.825,-35.919,447.408,175.280,15.897,152.345
C04793=1093.832,-35.669,447.396,175.282,15.898,152.345
C04794=1093.838,-35.419,447.384,175.284,15.899,152.345
C04795=1093.843,-35.170,447.372,175.286,15.901,152.345
C04796=1093.849,-34.920,447.359,175.288,15.902,152.345
C04797=1093.855,-34.670,447.347,175.290,15.902,152.345
C04798=1093.860,-34.421,447.334,175.291,15.904,152.344
C04799=1093.867,-34.172,447.322,175.293,15.905,152.344
C04800=1093.873,-33.922,447.310,175.295,15.906,152.344
C04801=1093.879,-33.672,447.297,175.296,15.907,152.344
C04802=1093.884,-33.423,447.285,175.298,15.908,152.344
C04803=1093.890,-33.173,447.273,175.300,15.909,152.344
C04804=1093.896,-32.904,447.259,175.301,15.910,152.344
C04805=1093.903,-32.636,447.246,175.304,15.911,152.343
C04806=1093.909,-32.366,447.233,175.305,15.912,152.343
C04807=1093.915,-32.097,447.219,175.307,15.914,152.343
C04808=1093.921,-31.847,447.207,175.309,15.915,152.343
C04809=1093.927,-31.598,447.195,175.311,15.915,152.343
C04810=1093.933,-31.348,447.182,175.312,15.917,152.343
C04811=1093.939,-31.098,447.170,175.314,15.918,152.343
C04812=1093.945,-30.849,447.157,175.316,15.920,152.342
C04813=1093.951,-30.600,447.144,175.318,15.920,152.342
C04814=1093.956,-30.350,447.132,175.320,15.921,152.342
C04815=1093.962,-30.100,447.119,175.321,15.923,152.342
C04816=1093.968,-29.850,447.106,175.323,15.923,152.342
C04817=1093.974,-29.601,447.094,175.325,15.924,152.342
C04818=1093.980,-29.351,447.082,175.326,15.926,152.342
C04819=1093.986,-29.102,447.069,175.328,15.927,152.341
C04820=1093.992,-28.852,447.056,175.330,15.927,152.341
C04821=1093.998,-28.602,447.044,175.331,15.929,152.341
C04822=1094.004,-28.353,447.032,175.334,15.930,152.341
C04823=1094.009,-28.103,447.019,175.335,15.931,152.341
C04824=1094.015,-27.853,447.007,175.337,15.932,152.341
C04825=1094.022,-27.604,446.993,175.339,15.933,152.340
C04826=1094.027,-27.354,446.981,175.341,15.934,152.340
C04827=1094.033,-27.104,446.968,175.342,15.935,152.340
C04828=1094.039,-26.855,446.956,175.344,15.936,152.340
C04829=1094.045,-26.606,446.943,175.346,15.937,152.340
C04830=1094.051,-26.356,446.930,175.347,15.939,152.340
C04831=1094.057,-26.106,446.918,175.349,15.940,152.340
C04832=1094.062,-25.857,446.905,175.351,15.941,152.339
C04833=1094.068,-25.608,446.892,175.353,15.942,152.339
C04834=1094.074,-25.358,446.880,175.355,15.943,152.339
C04835=1094.080,-25.108,446.867,175.356,15.944,152.339
C04836=1094.085,-24.858,446.854,175.358,15.945,152.339
C04837=1094.091,-24.609,446.841,175.360,15.946,152.339
C04838=1094.097,-24.359,446.828,175.361,15.947,152.339
C04839=1094.103,-24.109,446.816,175.363,15.949,152.339
C04840=1094.109,-23.859,446.803,175.365,15.950,152.338
C04841=1094.115,-23.610,446.790,175.367,15.951,152.338
C04842=1094.121,-23.360,446.778,175.369,15.952,152.338
C04843=1094.126,-23.111,446.765,175.370,15.953,152.338
C04844=1094.131,-22.861,446.751,175.372,15.955,152.338
C04845=1094.137,-22.612,446.739,175.374,15.955,152.338
C04846=1094.143,-22.362,446.726,175.376,15.956,152.338
C04847=1094.149,-22.112,446.713,175.377,15.958,152.337
C04848=1094.155,-21.863,446.701,175.380,15.959,152.337
C04849=1094.162,-21.613,446.687,175.381,15.960,152.337
C04850=1094.167,-21.364,446.675,175.383,15.961,152.337
C04851=1094.172,-21.114,446.662,175.385,15.962,152.337
C04852=1094.178,-20.865,446.649,175.386,15.963,152.337
C04853=1094.184,-20.615,446.636,175.388,15.964,152.336
C04854=1094.190,-20.365,446.623,175.390,15.965,152.336
C04855=1094.196,-20.116,446.610,175.392,15.967,152.336
C04856=1094.202,-19.866,446.598,175.394,15.968,152.336
C04857=1094.208,-19.616,446.584,175.396,15.969,152.336
C04858=1094.214,-19.366,446.571,175.397,15.970,152.336
C04859=1094.219,-19.118,446.558,175.399,15.971,152.336
C04860=1094.225,-18.868,446.546,175.400,15.972,152.336
C04861=1094.231,-18.619,446.533,175.402,15.973,152.335
C04862=1094.237,-18.369,446.520,175.405,15.975,152.335
C04863=1094.243,-18.119,446.506,175.406,15.976,152.335
C04864=1094.249,-17.869,446.494,175.408,15.977,152.335
C04865=1094.255,-17.619,446.481,175.410,15.978,152.335
C04866=1094.261,-17.370,446.468,175.411,15.979,152.335
C04867=1094.267,-17.120,446.455,175.413,15.980,152.335
C04868=1094.273,-16.851,446.441,175.416,15.981,152.334
C04869=1094.279,-16.581,446.427,175.417,15.983,152.334
C04870=1094.286,-16.311,446.412,175.419,15.984,152.334
C04871=1094.292,-16.041,446.398,175.422,15.985,152.334
C04872=1094.298,-15.792,446.385,175.423,15.986,152.334
C04873=1094.304,-15.542,446.372,175.425,15.987,152.334
C04874=1094.309,-15.292,446.359,175.426,15.989,152.333
C04875=1094.316,-15.043,446.346,175.428,15.989,152.333
C04876=1094.321,-14.793,446.333,175.430,15.990,152.333
C04877=1094.327,-14.543,446.319,175.432,15.992,152.333
C04878=1094.332,-14.294,446.307,175.434,15.993,152.333
C04879=1094.338,-14.045,446.294,175.436,15.994,152.333
C04880=1094.344,-13.795,446.280,175.437,15.995,152.332
C04881=1094.350,-13.546,446.267,175.439,15.996,152.332
C04882=1094.355,-13.296,446.253,175.440,15.997,152.332
C04883=1094.361,-13.046,446.241,175.443,15.999,152.332
C04884=1094.367,-12.797,446.228,175.445,16.000,152.332
C04885=1094.373,-12.547,446.214,175.446,16.001,152.332
C04886=1094.379,-12.297,446.201,175.448,16.002,152.332
C04887=1094.384,-12.048,446.187,175.450,16.003,152.331
C04888=1094.390,-11.798,446.174,175.451,16.004,152.331
C04889=1094.396,-11.549,446.162,175.454,16.006,152.331
C04890=1094.402,-11.299,446.148,175.455,16.007,152.331
C04891=1094.408,-11.050,446.134,175.457,16.008,152.331
C04892=1094.413,-10.800,446.121,175.459,16.009,152.331
C04893=1094.419,-10.550,446.108,175.461,16.010,152.331
C04894=1094.426,-10.301,446.095,175.462,16.011,152.331
C04895=1094.431,-10.051,446.082,175.465,16.012,152.330
C04896=1094.437,-9.802,446.068,175.466,16.014,152.330
C04897=1094.443,-9.552,446.054,175.468,16.015,152.330
C04898=1094.449,-9.303,446.041,175.470,16.016,152.330
C04899=1094.454,-9.053,446.028,175.472,16.017,152.330
C04900=1094.460,-8.803,446.015,175.474,16.018,152.330
C04901=1094.466,-8.554,446.001,175.476,16.019,152.329
C04902=1094.472,-8.304,445.988,175.477,16.020,152.329
C04903=1094.478,-8.055,445.975,175.479,16.021,152.329
C04904=1094.483,-7.805,445.961,175.481,16.022,152.329
C04905=1094.489,-7.556,445.948,175.483,16.024,152.329
C04906=1094.495,-7.306,445.934,175.485,16.025,152.329
C04907=1094.501,-7.056,445.921,175.486,16.026,152.329
C04908=1094.506,-6.807,445.908,175.488,16.027,152.328
C04909=1094.513,-6.557,445.894,175.490,16.028,152.328
C04910=1094.518,-6.308,445.880,175.492,16.029,152.328
C04911=1094.524,-6.059,445.867,175.494,16.031,152.328
C04912=1094.530,-5.808,445.853,175.496,16.031,152.328
C04913=1094.536,-5.558,445.840,175.497,16.033,152.328
C04914=1094.542,-5.309,445.827,175.499,16.034,152.327
C04915=1094.548,-5.060,445.813,175.501,16.034,152.327
C04916=1094.553,-4.810,445.799,175.503,16.036,152.327
C04917=1094.560,-4.561,445.786,175.505,16.037,152.327
C04918=1094.565,-4.311,445.772,175.507,16.038,152.327
C04919=1094.571,-4.062,445.759,175.508,16.039,152.327
C04920=1094.577,-3.812,445.745,175.510,16.040,152.327
C04921=1094.583,-3.562,445.733,175.513,16.042,152.326
C04922=1094.589,-3.312,445.718,175.514,16.043,152.326
C04923=1094.594,-3.063,445.705,175.516,16.044,152.326
C04924=1094.600,-2.813,445.691,175.518,16.045,152.326
C04925=1094.606,-2.564,445.677,175.519,16.046,152.326
C04926=1094.611,-2.314,445.664,175.522,16.048,152.326
C04927=1094.618,-2.065,445.650,175.523,16.049,152.325
C04928=1094.623,-1.815,445.636,175.525,16.050,152.325
C04929=1094.629,-1.566,445.623,175.527,16.051,152.325
C04930=1094.634,-1.316,445.609,175.529,16.052,152.325
C04931=1094.640,-1.067,445.595,175.531,16.053,152.325
C04932=1094.646,-0.796,445.581,175.533,16.054,152.325
C04933=1094.653,-0.524,445.566,175.535,16.056,152.324
C04934=1094.659,-0.253,445.551,175.537,16.057,152.324
C04935=1094.665,0.019,445.536,175.538,16.058,152.324
C04936=1094.671,0.269,445.522,175.541,16.060,152.324
C04937=1094.676,0.518,445.508,175.543,16.061,152.324
C04938=1094.682,0.768,445.494,175.544,16.062,152.324
C04939=1094.688,1.017,445.481,175.546,16.063,152.324
C04940=1094.693,1.267,445.467,175.549,16.064,152.323
C04941=1094.699,1.516,445.453,175.550,16.065,152.323
C04942=1094.704,1.766,445.439,175.552,16.066,152.323
C04943=1094.711,2.015,445.426,175.554,16.067,152.323
C04944=1094.717,2.265,445.412,175.556,16.069,152.323
C04945=1094.722,2.515,445.398,175.558,16.070,152.323
C04946=1094.728,2.765,445.384,175.560,16.071,152.322
C04947=1094.734,3.014,445.371,175.561,16.072,152.322
C04948=1094.740,3.263,445.356,175.563,16.073,152.322
C04949=1094.745,3.512,445.342,175.565,16.074,152.322
C04950=1094.751,3.762,445.328,175.567,16.076,152.322
C04951=1094.757,4.012,445.314,175.569,16.077,152.322
C04952=1094.763,4.261,445.301,175.570,16.077,152.322
C04953=1094.768,4.511,445.287,175.573,16.079,152.321
C04954=1094.774,4.761,445.273,175.574,16.080,152.321
C04955=1094.779,5.010,445.259,175.576,16.081,152.321
C04956=1094.786,5.260,445.244,175.578,16.082,152.321
C04957=1094.791,5.509,445.230,175.580,16.084,152.321
C04958=1094.797,5.759,445.217,175.582,16.085,152.321
C04959=1094.803,6.008,445.203,175.584,16.086,152.320
C04960=1094.808,6.258,445.189,175.586,16.086,152.320
C04961=1094.815,6.508,445.174,175.588,16.088,152.320
C04962=1094.820,6.757,445.161,175.590,16.089,152.320
C04963=1094.826,7.007,445.147,175.592,16.090,152.320
C04964=1094.832,7.256,445.133,175.593,16.091,152.320
C04965=1094.837,7.505,445.120,175.596,16.093,152.319
C04966=1094.844,7.755,445.105,175.598,16.094,152.319
C04967=1094.849,8.005,445.091,175.599,16.095,152.319
C04968=1094.855,8.254,445.077,175.601,16.096,152.319
C04969=1094.860,8.504,445.063,175.603,16.097,152.319
C04970=1094.867,8.754,445.048,175.605,16.098,152.319
C04971=1094.873,9.003,445.035,175.607,16.099,152.318
C04972=1094.878,9.252,445.021,175.608,16.100,152.318
C04973=1094.884,9.501,445.006,175.611,16.102,152.318
C04974=1094.890,9.752,444.992,175.613,16.103,152.318
C04975=1094.896,10.001,444.978,175.615,16.103,152.318
C04976=1094.901,10.250,444.964,175.616,16.105,152.318
C04977=1094.907,10.500,444.949,175.619,16.106,152.317
C04978=1094.913,10.750,444.936,175.621,16.107,152.317
C04979=1094.919,10.999,444.922,175.622,16.108,152.317
C04980=1094.925,11.248,444.908,175.624,16.109,152.317
C04981=1094.931,11.498,444.894,175.626,16.111,152.317
C04982=1094.937,11.747,444.879,175.628,16.111,152.316
C04983=1094.942,11.997,444.865,175.630,16.112,152.316
C04984=1094.948,12.247,444.851,175.632,16.114,152.316
C04985=1094.954,12.496,444.836,175.634,16.115,152.316
C04986=1094.960,12.746,444.822,175.636,16.116,152.316
C04987=1094.966,12.995,444.807,175.638,16.117,152.316
C04988=1094.971,13.245,444.794,175.639,16.118,152.316
C04989=1094.977,13.495,444.780,175.642,16.119,152.315
C04990=1094.983,13.744,444.765,175.644,16.120,152.315
C04991=1094.989,13.994,444.751,175.645,16.121,152.315
C04992=1094.995,14.243,444.737,175.648,16.123,152.315
C04993=1095.001,14.493,444.723,175.650,16.123,152.314
C04994=1095.006,14.742,444.708,175.651,16.125,152.314
C04995=1095.012,14.992,444.694,175.653,16.125,152.314
C04996=1095.018,15.265,444.678,175.656,16.127,152.314
C04997=1095.024,15.538,444.663,175.658,16.128,152.314
C04998=1095.031,15.812,444.646,175.660,16.129,152.314
C04999=1095.038,16.085,444.630,175.662,16.131,152.314
C05000=1095.043,16.335,444.616,175.664,16.132,152.313
C05001=1095.049,16.584,444.602,175.666,16.133,152.313
C05002=1095.055,16.834,444.588,175.668,16.134,152.313
C05003=1095.061,17.083,444.573,175.670,16.135,152.313
C05004=1095.066,17.333,444.559,175.672,16.136,152.312
C05005=1095.072,17.583,444.544,175.674,16.137,152.312
C05006=1095.077,17.832,444.530,175.676,16.138,152.312
C05007=1095.084,18.082,444.515,175.678,16.140,152.312
C05008=1095.089,18.331,444.500,175.680,16.140,152.312
C05009=1095.095,18.580,444.486,175.681,16.142,152.312
C05010=1095.101,18.830,444.471,175.684,16.143,152.311
C05011=1095.107,19.080,444.458,175.686,16.144,152.311
C05012=1095.112,19.329,444.442,175.688,16.145,152.311
C05013=1095.118,19.578,444.427,175.689,16.146,152.311
C05014=1095.124,19.828,444.414,175.692,16.147,152.311
C05015=1095.130,20.078,444.399,175.693,16.148,152.311
C05016=1095.136,20.327,444.385,175.695,16.149,152.310
C05017=1095.141,20.576,444.370,175.698,16.151,152.310
C05018=1095.147,20.826,444.355,175.700,16.151,152.310
C05019=1095.152,21.076,444.341,175.701,16.153,152.310
C05020=1095.158,21.325,444.326,175.704,16.154,152.310
C05021=1095.165,21.574,444.311,175.706,16.155,152.309
C05022=1095.169,21.824,444.297,175.707,16.156,152.309
C05023=1095.176,22.074,444.282,175.709,16.157,152.309
C05024=1095.181,22.323,444.267,175.711,16.159,152.309
C05025=1095.187,22.572,444.253,175.713,16.159,152.309
C05026=1095.193,22.822,444.238,175.715,16.160,152.308
C05027=1095.198,23.071,444.223,175.718,16.162,152.308
C05028=1095.205,23.321,444.208,175.720,16.162,152.308
C05029=1095.209,23.571,444.194,175.721,16.164,152.308
C05030=1095.215,23.820,444.179,175.724,16.165,152.308
C05031=1095.222,24.070,444.164,175.725,16.166,152.308
C05032=1095.227,24.318,444.150,175.727,16.167,152.307
C05033=1095.233,24.569,444.135,175.730,16.168,152.307
C05034=1095.239,24.818,444.120,175.732,16.169,152.307
C05035=1095.245,25.068,444.105,175.733,16.170,152.307
C05036=1095.250,25.317,444.090,175.735,16.171,152.307
C05037=1095.256,25.567,444.076,175.737,16.173,152.306
C05038=1095.262,25.816,444.061,175.739,16.173,152.306
C05039=1095.267,26.065,444.046,175.741,16.174,152.306
C05040=1095.273,26.315,444.031,175.744,16.176,152.306
C05041=1095.279,26.564,444.017,175.746,16.176,152.306
C05042=1095.285,26.814,444.001,175.747,16.178,152.305
C05043=1095.290,27.064,443.987,175.750,16.179,152.305
C05044=1095.297,27.313,443.972,175.752,16.180,152.305
C05045=1095.302,27.563,443.957,175.753,16.181,152.305
C05046=1095.308,27.812,443.942,175.756,16.182,152.305
C05047=1095.314,28.061,443.928,175.758,16.183,152.304
C05048=1095.319,28.311,443.912,175.759,16.184,152.304
C05049=1095.325,28.560,443.898,175.762,16.185,152.304
C05050=1095.331,28.810,443.882,175.764,16.186,152.304
C05051=1095.336,29.060,443.868,175.766,16.187,152.304
C05052=1095.343,29.309,443.853,175.768,16.189,152.303
C05053=1095.348,29.559,443.838,175.770,16.189,152.303
C05054=1095.354,29.808,443.823,175.772,16.191,152.303
C05055=1095.359,30.057,443.808,175.774,16.192,152.303
C05056=1095.366,30.307,443.793,175.776,16.193,152.303
C05057=1095.371,30.556,443.778,175.778,16.194,152.302
C05058=1095.377,30.806,443.763,175.780,16.195,152.302
C05059=1095.382,31.055,443.748,175.782,16.196,152.302
C05060=1095.389,31.331,443.731,175.785,16.197,152.302
C05061=1095.395,31.605,443.714,175.787,16.198,152.302
C05062=1095.401,31.880,443.698,175.789,16.200,152.301
C05063=1095.407,32.155,443.682,175.791,16.201,152.301
C05064=1095.414,32.405,443.667,175.794,16.202,152.301
C05065=1095.419,32.654,443.651,175.795,16.203,152.301
C05066=1095.425,32.903,443.636,175.797,16.204,152.301
C05067=1095.430,33.152,443.621,175.800,16.205,152.300
C05068=1095.436,33.402,443.605,175.801,16.206,152.300
C05069=1095.442,33.651,443.591,175.803,16.207,152.300
C05070=1095.447,33.901,443.575,175.806,16.208,152.300
C05071=1095.453,34.150,443.560,175.808,16.209,152.300
C05072=1095.459,34.400,443.545,175.809,16.210,152.299
C05073=1095.465,34.650,443.530,175.812,16.211,152.299
C05074=1095.470,34.899,443.515,175.814,16.212,152.299
C05075=1095.477,35.149,443.500,175.816,16.213,152.299
C05076=1095.482,35.398,443.485,175.818,16.214,152.298
C05077=1095.488,35.648,443.470,175.820,16.215,152.298
C05078=1095.493,35.896,443.454,175.822,16.216,152.298
C05079=1095.499,36.146,443.438,175.825,16.217,152.298
C05080=1095.505,36.396,443.423,175.826,16.218,152.297
C05081=1095.510,36.645,443.408,175.829,16.220,152.297
C05082=1095.517,36.895,443.393,175.831,16.221,152.297
C05083=1095.522,37.144,443.378,175.833,16.221,152.297
C05084=1095.528,37.393,443.362,175.835,16.222,152.297
C05085=1095.534,37.643,443.347,175.837,16.224,152.296
C05086=1095.539,37.892,443.332,175.839,16.224,152.296
C05087=1095.546,38.142,443.317,175.841,16.226,152.296
C05088=1095.551,38.392,443.301,175.843,16.227,152.296
C05089=1095.557,38.641,443.285,175.845,16.227,152.296
C05090=1095.562,38.891,443.270,175.848,16.229,152.295
C05091=1095.568,39.139,443.255,175.849,16.230,152.295
C05092=1095.574,39.389,443.240,175.852,16.231,152.295
C05093=1095.580,39.639,443.223,175.854,16.232,152.295
C05094=1095.585,39.888,443.208,175.856,16.233,152.294
C05095=1095.591,40.138,443.193,175.858,16.234,152.294
C05096=1095.596,40.387,443.178,175.860,16.235,152.294
C05097=1095.602,40.636,443.162,175.862,16.236,152.294
C05098=1095.608,40.886,443.146,175.865,16.237,152.294
C05099=1095.614,41.135,443.132,175.866,16.238,152.293
C05100=1095.619,41.385,443.116,175.869,16.239,152.293
C05101=1095.625,41.635,443.100,175.871,16.240,152.293
C05102=1095.630,41.884,443.085,175.873,16.241,152.293
C05103=1095.637,42.134,443.070,175.875,16.242,152.292
C05104=1095.642,42.383,443.053,175.877,16.243,152.292
C05105=1095.648,42.632,443.038,175.879,16.244,152.292
C05106=1095.653,42.881,443.022,175.882,16.245,152.292
C05107=1095.659,43.131,443.006,175.883,16.246,152.291
C05108=1095.665,43.380,442.992,175.886,16.248,152.291
C05109=1095.671,43.630,442.976,175.888,16.248,152.291
C05110=1095.677,43.880,442.960,175.890,16.249,152.291
C05111=1095.682,44.129,442.945,175.892,16.250,152.291
C05112=1095.687,44.378,442.929,175.894,16.251,152.290
C05113=1095.693,44.628,442.913,175.896,16.252,152.290
C05114=1095.698,44.877,442.897,175.898,16.253,152.290
C05115=1095.704,45.127,442.882,175.900,16.254,152.290
C05116=1095.709,45.376,442.866,175.903,16.255,152.289
C05117=1095.715,45.626,442.850,175.905,16.256,152.289
C05118=1095.721,45.875,442.835,175.907,16.257,152.289
C05119=1095.726,46.124,442.819,175.909,16.258,152.289
C05120=1095.732,46.374,442.803,175.911,16.259,152.289
C05121=1095.738,46.623,442.787,175.914,16.261,152.288
C05122=1095.743,46.873,442.772,175.915,16.262,152.288
C05123=1095.749,47.122,442.756,175.917,16.262,152.288
C05124=1095.756,47.397,442.738,175.920,16.263,152.288
C05125=1095.762,47.672,442.721,175.923,16.265,152.287
C05126=1095.767,47.947,442.704,175.925,16.265,152.287
C05127=1095.774,48.222,442.687,175.927,16.267,152.287
C05128=1095.780,48.471,442.670,175.929,16.267,152.287
C05129=1095.785,48.721,442.655,175.932,16.269,152.286
C05130=1095.791,48.970,442.639,175.933,16.270,152.286
C05131=1095.796,49.219,442.623,175.936,16.271,152.286
C05132=1095.802,49.469,442.607,175.938,16.272,152.286
C05133=1095.807,49.718,442.591,175.940,16.272,152.285
C05134=1095.813,49.968,442.576,175.943,16.274,152.285
C05135=1095.819,50.217,442.559,175.944,16.274,152.285
C05136=1095.825,50.467,442.544,175.947,16.276,152.285
C05137=1095.831,50.716,442.528,175.949,16.277,152.284
C05138=1095.836,50.965,442.512,175.951,16.278,152.284
C05139=1095.842,51.215,442.496,175.953,16.279,152.284
C05140=1095.848,51.464,442.480,175.955,16.280,152.284
C05141=1095.854,51.714,442.464,175.958,16.281,152.283
C05142=1095.859,51.963,442.448,175.960,16.281,152.283
C05143=1095.865,52.212,442.432,175.963,16.283,152.283
C05144=1095.870,52.462,442.416,175.964,16.283,152.283
C05145=1095.876,52.712,442.400,175.966,16.284,152.282
C05146=1095.882,52.961,442.384,175.969,16.285,152.282
C05147=1095.887,53.210,442.368,175.971,16.286,152.282
C05148=1095.892,53.460,442.352,175.974,16.287,152.282
C05149=1095.898,53.709,442.336,175.975,16.288,152.281
C05150=1095.904,53.959,442.320,175.977,16.289,152.281
C05151=1095.910,54.208,442.303,175.980,16.290,152.281
C05152=1095.915,54.457,442.288,175.982,16.291,152.281
C05153=1095.921,54.707,442.272,175.985,16.292,152.280
C05154=1095.927,54.956,442.256,175.987,16.293,152.280
C05155=1095.933,55.205,442.239,175.989,16.294,152.280
C05156=1095.939,55.455,442.224,175.991,16.295,152.279
C05157=1095.945,55.705,442.208,175.993,16.295,152.279
C05158=1095.950,55.954,442.191,175.996,16.297,152.279
C05159=1095.955,56.203,442.175,175.998,16.297,152.279
C05160=1095.961,56.452,442.159,176.000,16.299,152.278
C05161=1095.967,56.702,442.142,176.002,16.299,152.278
C05162=1095.973,56.952,442.127,176.004,16.300,152.278
C05163=1095.979,57.201,442.111,176.007,16.301,152.278
C05164=1095.985,57.450,442.094,176.009,16.302,152.277
C05165=1095.990,57.700,442.077,176.011,16.303,152.277
C05166=1095.996,57.949,442.061,176.013,16.304,152.277
C05167=1096.002,58.199,442.045,176.016,16.305,152.277
C05168=1096.008,58.448,442.029,176.018,16.306,152.276
C05169=1096.013,58.697,442.013,176.020,16.306,152.276
C05170=1096.019,58.947,441.997,176.023,16.307,152.276
C05171=1096.024,59.196,441.980,176.025,16.308,152.275
C05172=1096.030,59.446,441.964,176.027,16.309,152.275
C05173=1096.036,59.695,441.948,176.029,16.310,152.275
C05174=1096.042,59.944,441.932,176.032,16.311,152.275
C05175=1096.048,60.194,441.915,176.034,16.312,152.274
C05176=1096.054,60.443,441.899,176.036,16.313,152.274
C05177=1096.059,60.693,441.882,176.038,16.314,152.274
C05178=1096.065,60.942,441.866,176.040,16.314,152.273
C05179=1096.071,61.191,441.850,176.043,16.315,152.273
C05180=1096.077,61.441,441.833,176.045,16.316,152.273
C05181=1096.083,61.690,441.817,176.048,16.317,152.273
C05182=1096.088,61.940,441.800,176.050,16.318,152.272
C05183=1096.094,62.189,441.784,176.053,16.319,152.272
C05184=1096.100,62.438,441.768,176.055,16.319,152.272
C05185=1096.106,62.688,441.752,176.056,16.320,152.271
C05186=1096.111,62.937,441.735,176.059,16.321,152.271
C05187=1096.117,63.187,441.718,176.061,16.322,152.271
C05188=1096.123,63.461,441.700,176.064,16.323,152.270
C05189=1096.130,63.736,441.683,176.067,16.324,152.270
C05190=1096.137,64.011,441.664,176.069,16.325,152.270
C05191=1096.143,64.285,441.646,176.072,16.326,152.269
C05192=1096.149,64.534,441.629,176.073,16.326,152.269
C05193=1096.154,64.784,441.612,176.076,16.328,152.269
C05194=1096.160,65.033,441.596,176.078,16.328,152.269
C05195=1096.166,65.283,441.580,176.081,16.329,152.268
C05196=1096.171,65.532,441.563,176.083,16.330,152.268
C05197=1096.177,65.782,441.547,176.086,16.331,152.268
C05198=1096.182,66.031,441.530,176.087,16.332,152.267
C05199=1096.189,66.280,441.513,176.090,16.333,152.267
C05200=1096.195,66.530,441.497,176.092,16.333,152.267
C05201=1096.200,66.779,441.480,176.095,16.335,152.267
C05202=1096.206,67.029,441.464,176.097,16.335,152.266
C05203=1096.211,67.278,441.447,176.100,16.337,152.266
C05204=1096.217,67.527,441.430,176.102,16.337,152.266
C05205=1096.222,67.777,441.413,176.104,16.337,152.265
C05206=1096.228,68.026,441.397,176.106,16.339,152.265
C05207=1096.234,68.276,441.380,176.108,16.339,152.265
C05208=1096.240,68.525,441.364,176.111,16.340,152.264
C05209=1096.245,68.774,441.346,176.113,16.341,152.264
C05210=1096.251,69.023,441.330,176.116,16.342,152.264
C05211=1096.257,69.273,441.313,176.118,16.342,152.263
C05212=1096.262,69.522,441.297,176.121,16.344,152.263
C05213=1096.268,69.771,441.280,176.123,16.344,152.263
C05214=1096.274,70.021,441.263,176.125,16.346,152.263
C05215=1096.279,70.270,441.246,176.127,16.346,152.262
C05216=1096.285,70.519,441.229,176.130,16.347,152.262
C05217=1096.290,70.769,441.212,176.132,16.348,152.262
C05218=1096.296,71.018,441.196,176.134,16.348,152.261
C05219=1096.302,71.267,441.178,176.137,16.349,152.261
C05220=1096.308,71.516,441.162,176.139,16.350,152.261
C05221=1096.313,71.766,441.145,176.142,16.351,152.260
C05222=1096.318,72.015,441.128,176.144,16.352,152.260
C05223=1096.325,72.265,441.111,176.146,16.353,152.260
C05224=1096.330,72.515,441.094,176.149,16.353,152.259
C05225=1096.336,72.764,441.077,176.151,16.354,152.259
C05226=1096.342,73.013,441.060,176.153,16.355,152.259
C05227=1096.347,73.263,441.044,176.156,16.356,152.258
C05228=1096.353,73.512,441.027,176.158,16.357,152.258
C05229=1096.358,73.761,441.010,176.161,16.358,152.258
C05230=1096.364,74.010,440.992,176.163,16.358,152.258
C05231=1096.370,74.260,440.976,176.166,16.359,152.257
C05232=1096.375,74.509,440.958,176.167,16.360,152.257
C05233=1096.381,74.758,440.941,176.170,16.361,152.257
C05234=1096.387,75.008,440.924,176.172,16.361,152.256
C05235=1096.393,75.258,440.907,176.175,16.362,152.256
C05236=1096.398,75.507,440.890,176.177,16.363,152.256
C05237=1096.404,75.756,440.873,176.180,16.364,152.255
C05238=1096.409,76.006,440.857,176.182,16.364,152.255
C05239=1096.415,76.255,440.839,176.185,16.366,152.255
C05240=1096.421,76.503,440.822,176.187,16.366,152.254
C05241=1096.427,76.754,440.805,176.190,16.367,152.254
C05242=1096.432,77.003,440.787,176.192,16.367,152.254
C05243=1096.438,77.252,440.771,176.194,16.368,152.253
C05244=1096.444,77.501,440.753,176.197,16.369,152.253
C05245=1096.449,77.751,440.737,176.199,16.370,152.253
C05246=1096.455,78.000,440.719,176.202,16.370,152.252
C05247=1096.461,78.250,440.702,176.203,16.371,152.252
C05248=1096.467,78.499,440.685,176.206,16.372,152.252
C05249=1096.472,78.748,440.667,176.208,16.373,152.251
C05250=1096.477,78.998,440.650,176.211,16.374,152.251
C05251=1096.484,79.246,440.633,176.213,16.374,152.251
C05252=1096.489,79.521,440.614,176.216,16.375,152.250
C05253=1096.496,79.796,440.595,176.219,16.376,152.250
C05254=1096.502,80.071,440.576,176.222,16.377,152.249
C05255=1096.509,80.345,440.557,176.224,16.378,152.249
C05256=1096.514,80.595,440.540,176.227,16.379,152.249
C05257=1096.519,80.844,440.522,176.229,16.379,152.249
C05258=1096.525,81.093,440.505,176.232,16.380,152.248
C05259=1096.530,81.342,440.488,176.233,16.381,152.248
C05260=1096.536,81.592,440.470,176.236,16.382,152.247
C05261=1096.542,81.841,440.453,176.238,16.382,152.247
C05262=1096.548,82.091,440.436,176.241,16.383,152.247
C05263=1096.553,82.340,440.419,176.243,16.384,152.247
C05264=1096.559,82.589,440.401,176.246,16.385,152.246
C05265=1096.565,82.838,440.383,176.249,16.385,152.246
C05266=1096.570,83.088,440.366,176.251,16.386,152.245
C05267=1096.576,83.337,440.349,176.254,16.387,152.245
C05268=1096.581,83.586,440.331,176.256,16.388,152.245
C05269=1096.587,83.836,440.313,176.259,16.388,152.244
C05270=1096.592,84.086,440.296,176.261,16.389,152.244
C05271=1096.598,84.335,440.279,176.264,16.390,152.244
C05272=1096.603,84.584,440.261,176.266,16.390,152.243
C05273=1096.610,84.833,440.243,176.269,16.391,152.243
C05274=1096.615,85.082,440.226,176.271,16.392,152.243
C05275=1096.621,85.331,440.209,176.274,16.392,152.242
C05276=1096.627,85.581,440.192,176.276,16.393,152.242
C05277=1096.633,85.831,440.174,176.279,16.394,152.241
C05278=1096.638,86.080,440.157,176.281,16.395,152.241
C05279=1096.644,86.329,440.139,176.284,16.395,152.241
C05280=1096.650,86.578,440.121,176.286,16.396,152.240
C05281=1096.655,86.827,440.103,176.288,16.397,152.240
C05282=1096.661,87.076,440.086,176.291,16.397,152.240
C05283=1096.667,87.326,440.068,176.294,16.398,152.239
C05284=1096.672,87.576,440.051,176.296,16.398,152.239
C05285=1096.678,87.825,440.034,176.298,16.400,152.239
C05286=1096.684,88.075,440.016,176.301,16.400,152.238
C05287=1096.689,88.324,439.998,176.304,16.401,152.238
C05288=1096.695,88.573,439.980,176.306,16.401,152.238
C05289=1096.701,88.822,439.963,176.308,16.402,152.237
C05290=1096.707,89.071,439.945,176.311,16.402,152.237
C05291=1096.712,89.320,439.927,176.314,16.403,152.236
C05292=1096.718,89.570,439.909,176.316,16.404,152.236
C05293=1096.724,89.819,439.892,176.319,16.405,152.236
C05294=1096.729,90.068,439.874,176.321,16.405,152.235
C05295=1096.735,90.318,439.856,176.324,16.406,152.235
C05296=1096.741,90.567,439.839,176.327,16.406,152.234
C05297=1096.746,90.817,439.820,176.329,16.407,152.234
C05298=1096.752,91.066,439.803,176.332,16.408,152.234
C05299=1096.757,91.315,439.785,176.334,16.408,152.233
C05300=1096.763,91.565,439.767,176.337,16.409,152.233
C05301=1096.769,91.814,439.750,176.339,16.410,152.233
C05302=1096.775,92.062,439.731,176.342,16.411,152.232
C05303=1096.780,92.312,439.713,176.344,16.411,152.232
C05304=1096.786,92.562,439.695,176.347,16.412,152.231
C05305=1096.791,92.811,439.678,176.349,16.412,152.231
C05306=1096.797,93.060,439.660,176.352,16.413,152.231
C05307=1096.803,93.309,439.642,176.354,16.413,152.230
C05308=1096.808,93.559,439.624,176.357,16.414,152.230
C05309=1096.814,93.808,439.606,176.360,16.415,152.229
C05310=1096.819,94.057,439.589,176.362,16.416,152.229
C05311=1096.826,94.307,439.570,176.365,16.416,152.229
C05312=1096.830,94.556,439.552,176.367,16.417,152.228
C05313=1096.836,94.805,439.534,176.370,16.417,152.228
C05314=1096.842,95.055,439.516,176.372,16.418,152.227
C05315=1096.848,95.304,439.499,176.375,16.419,152.227
C05316=1096.854,95.579,439.478,176.378,16.419,152.227
C05317=1096.860,95.853,439.459,176.380,16.420,152.226
C05318=1096.867,96.128,439.438,176.383,16.420,152.226
C05319=1096.873,96.402,439.418,176.386,16.421,152.225
C05320=1096.879,96.652,439.401,176.389,16.422,152.225
C05321=1096.883,96.901,439.382,176.391,16.422,152.225
C05322=1096.889,97.150,439.365,176.394,16.423,152.224
C05323=1096.895,97.399,439.346,176.396,16.423,152.224
C05324=1096.901,97.648,439.329,176.399,16.424,152.223
C05325=1096.906,97.898,439.310,176.401,16.425,152.223
C05326=1096.912,98.147,439.292,176.404,16.426,152.223
C05327=1096.918,98.396,439.274,176.406,16.426,152.222
C05328=1096.923,98.646,439.256,176.409,16.427,152.222
C05329=1096.929,98.895,439.237,176.412,16.427,152.221
C05330=1096.935,99.144,439.219,176.415,16.428,152.221
C05331=1096.940,99.394,439.201,176.417,16.429,152.220
C05332=1096.946,99.642,439.183,176.420,16.429,152.220
C05333=1096.952,99.892,439.165,176.423,16.430,152.220
C05334=1096.957,100.142,439.147,176.425,16.430,152.219
C05335=1096.963,100.391,439.128,176.428,16.431,152.219
C05336=1096.969,100.640,439.110,176.430,16.431,152.218
C05337=1096.975,100.889,439.091,176.433,16.432,152.218
C05338=1096.980,101.138,439.074,176.435,16.432,152.218
C05339=1096.986,101.388,439.056,176.438,16.432,152.217
C05340=1096.991,101.637,439.037,176.441,16.434,152.217
C05341=1096.998,101.886,439.019,176.443,16.434,152.216
C05342=1097.003,102.135,439.000,176.446,16.435,152.216
C05343=1097.009,102.385,438.982,176.448,16.435,152.216
C05344=1097.014,102.634,438.963,176.451,16.436,152.215
C05345=1097.020,102.883,438.945,176.454,16.436,152.215
C05346=1097.025,103.132,438.926,176.457,16.436,152.214
C05347=1097.031,103.382,438.908,176.460,16.437,152.214
C05348=1097.036,103.631,438.889,176.462,16.437,152.213
C05349=1097.042,103.880,438.872,176.465,16.438,152.213
C05350=1097.048,104.130,438.852,176.467,16.438,152.212
C05351=1097.053,104.379,438.834,176.470,16.439,152.212
C05352=1097.059,104.628,438.816,176.472,16.439,152.212
C05353=1097.064,104.878,438.797,176.475,16.440,152.211
C05354=1097.070,105.127,438.779,176.478,16.441,152.211
C05355=1097.075,105.376,438.761,176.480,16.441,152.210
C05356=1097.082,105.625,438.742,176.483,16.442,152.210
C05357=1097.087,105.874,438.723,176.486,16.442,152.210
C05358=1097.093,106.124,438.705,176.489,16.443,152.209
C05359=1097.099,106.373,438.686,176.491,16.443,152.209
C05360=1097.103,106.622,438.668,176.494,16.444,152.208
C05361=1097.110,106.872,438.649,176.497,16.445,152.208
C05362=1097.115,107.120,438.630,176.499,16.445,152.207
C05363=1097.121,107.370,438.612,176.502,16.446,152.207
C05364=1097.127,107.619,438.593,176.504,16.446,152.206
C05365=1097.132,107.868,438.575,176.508,16.446,152.206
C05366=1097.138,108.118,438.556,176.511,16.447,152.205
C05367=1097.143,108.367,438.537,176.513,16.447,152.205
C05368=1097.149,108.616,438.519,176.516,16.448,152.205
C05369=1097.155,108.866,438.500,176.518,16.448,152.204
C05370=1097.161,109.114,438.482,176.521,16.449,152.204
C05371=1097.166,109.364,438.463,176.523,16.449,152.203
C05372=1097.172,109.613,438.443,176.526,16.450,152.203
C05373=1097.177,109.862,438.426,176.529,16.451,152.202
C05374=1097.183,110.112,438.407,176.532,16.450,152.202
C05375=1097.189,110.361,438.387,176.535,16.451,152.201
C05376=1097.195,110.609,438.369,176.537,16.451,152.201
C05377=1097.200,110.859,438.350,176.540,16.452,152.200
C05378=1097.206,111.109,438.331,176.543,16.453,152.200
C05379=1097.212,111.357,438.313,176.545,16.453,152.200
C05380=1097.217,111.633,438.292,176.549,16.453,152.199
C05381=1097.224,111.907,438.271,176.552,16.454,152.199
C05382=1097.230,112.182,438.250,176.555,16.454,152.198
C05383=1097.237,112.456,438.229,176.558,16.455,152.198
C05384=1097.242,112.705,438.210,176.560,16.455,152.197
C05385=1097.248,112.954,438.191,176.563,16.456,152.197
C05386=1097.254,113.204,438.173,176.566,16.456,152.196
C05387=1097.259,113.453,438.154,176.569,16.456,152.196
C05388=1097.265,113.702,438.135,176.572,16.457,152.195
C05389=1097.270,113.952,438.116,176.574,16.458,152.195
C05390=1097.277,114.201,438.097,176.577,16.458,152.194
C05391=1097.282,114.450,438.078,176.579,16.458,152.194
C05392=1097.287,114.699,438.059,176.582,16.459,152.193
C05393=1097.293,114.948,438.040,176.586,16.459,152.193
C05394=1097.298,115.197,438.021,176.588,16.460,152.192
C05395=1097.304,115.447,438.002,176.591,16.460,152.192
C05396=1097.310,115.696,437.983,176.593,16.461,152.192
C05397=1097.315,115.945,437.964,176.596,16.461,152.191
C05398=1097.320,116.194,437.944,176.599,16.462,152.191
C05399=1097.326,116.444,437.925,176.601,16.462,152.190
C05400=1097.331,116.692,437.906,176.605,16.462,152.190
C05401=1097.338,116.942,437.888,176.607,16.463,152.189
C05402=1097.343,117.191,437.868,176.610,16.463,152.189
C05403=1097.349,117.440,437.849,176.613,16.464,152.188
C05404=1097.354,117.689,437.830,176.615,16.464,152.188
C05405=1097.360,117.939,437.811,176.618,16.464,152.187
C05406=1097.365,118.188,437.792,176.621,16.465,152.187
C05407=1097.371,118.437,437.773,176.624,16.466,152.186
C05408=1097.376,118.686,437.754,176.627,16.466,152.186
C05409=1097.382,118.936,437.734,176.629,16.466,152.185
C05410=1097.388,119.185,437.715,176.632,16.467,152.185
C05411=1097.393,119.434,437.696,176.635,16.467,152.184
C05412=1097.398,119.683,437.677,176.638,16.467,152.184
C05413=1097.404,119.933,437.658,176.641,16.468,152.183
C05414=1097.410,120.181,437.638,176.643,16.468,152.183
C05415=1097.416,120.431,437.619,176.646,16.469,152.183
C05416=1097.421,120.680,437.600,176.649,16.469,152.182
C05417=1097.426,120.929,437.581,176.652,16.469,152.182
C05418=1097.432,121.178,437.561,176.655,16.470,152.181
C05419=1097.438,121.428,437.542,176.657,16.470,152.181
C05420=1097.444,121.677,437.522,176.660,16.470,152.180
C05421=1097.449,121.925,437.503,176.663,16.471,152.180
C05422=1097.455,122.175,437.484,176.666,16.471,152.179
C05423=1097.460,122.424,437.465,176.669,16.472,152.179
C05424=1097.466,122.673,437.444,176.672,16.472,152.178
C05425=1097.471,122.923,437.425,176.674,16.472,152.178
C05426=1097.477,123.172,437.406,176.678,16.473,152.177
C05427=1097.483,123.422,437.386,176.680,16.473,152.177
C05428=1097.488,123.670,437.367,176.683,16.473,152.176
C05429=1097.494,123.919,437.348,176.686,16.474,152.175
C05430=1097.499,124.169,437.328,176.688,16.474,152.175
C05431=1097.505,124.418,437.308,176.692,16.474,152.174
C05432=1097.511,124.667,437.289,176.695,16.475,152.174
C05433=1097.517,124.916,437.270,176.697,16.475,152.174
C05434=1097.523,125.165,437.250,176.700,16.475,152.173
C05435=1097.528,125.415,437.231,176.703,16.476,152.173
C05436=1097.534,125.663,437.212,176.706,16.476,152.172
C05437=1097.539,125.912,437.191,176.709,16.476,152.171
C05438=1097.544,126.162,437.172,176.711,16.476,152.171
C05439=1097.550,126.411,437.153,176.715,16.477,152.170
C05440=1097.556,126.660,437.133,176.718,16.477,152.170
C05441=1097.562,126.910,437.114,176.720,16.477,152.169
C05442=1097.568,127.158,437.094,176.723,16.478,152.169
C05443=1097.574,127.408,437.074,176.726,16.478,152.168
C05444=1097.580,127.682,437.053,176.729,16.478,152.168
C05445=1097.586,127.957,437.031,176.732,16.478,152.167
C05446=1097.592,128.232,437.010,176.735,16.479,152.167
C05447=1097.599,128.507,436.988,176.739,16.479,152.166
C05448=1097.605,128.756,436.968,176.742,16.479,152.165
C05449=1097.610,129.004,436.949,176.744,16.479,152.165
C05450=1097.615,129.254,436.928,176.747,16.480,152.164
C05451=1097.621,129.502,436.908,176.751,16.480,152.164
C05452=1097.627,129.752,436.889,176.753,16.480,152.163
C05453=1097.633,130.001,436.869,176.756,16.481,152.163
